LIN {X 0,Y 256.905,Z 476.365,A -85,B 0,C 180,E1 -19492.497,E2 -19492.497} C_VEL
LIN {X 0,Y 253.744,Z 490.842,A -85,B 0,C 180,E1 -19494.195,E2 -19494.195} C_VEL
LIN {X 0,Y 250.282,Z 505.582,A -85,B 0,C 180,E1 -19496.323,E2 -19496.323} C_VEL
LIN {X 0,Y 246.869,Z 518.814,A -85,B 0,C 180,E1 -19498.654,E2 -19498.654} C_VEL
LIN {X 0,Y 243.85,Z 530.517,A -85,B 0,C 180,E1 -19501.14,E2 -19501.14} C_VEL
LIN {X 0,Y 240.923,Z 541.947,A -85,B 0,C 180,E1 -19504.056,E2 -19504.056} C_VEL
LIN {X 0,Y 238.58,Z 551.642,A -85,B 0,C 180,E1 -19507.031,E2 -19507.031} C_VEL
LIN {X 0,Y 236.824,Z 559.89,A -85,B 0,C 180,E1 -19510.05,E2 -19510.05} C_VEL
LIN {X 0,Y 235.764,Z 565.839,A -85,B 0,C 180,E1 -19512.662,E2 -19512.662} C_VEL
LIN {X 0,Y 234.817,Z 572.47,A -85,B 0,C 180,E1 -19516.151,E2 -19516.151} C_VEL
LIN {X 0,Y 234.44,Z 577.709,A -85,B 0,C 180,E1 -19519.642,E2 -19519.642} C_VEL
LIN {X 0,Y 234.502,Z 581.558,A -85,B 0,C 180,E1 -19523.119,E2 -19523.119} C_VEL
LIN {X 0,Y 234.607,Z 584.124,A -85,B 0,C 180,E1 -19526.569,E2 -19526.569} C_VEL
LIN {X 0,Y 234.696,Z 584.956,A -85,B 0,C 180,E1 -19528.288,E2 -19528.288} C_VEL
LIN {X 0,Y 234.734,Z 585.482,A -85,B 0,C 180,E1 -19530.004,E2 -19530.004} C_VEL
LIN {X 0,Y 234.443,Z 585.509,A -85,B 0,C 180,E1 -19533.441,E2 -19533.441} C_VEL
LIN {X 0,Y 234.354,Z 585.124,A -85,B 0,C 180,E1 -19535.166,E2 -19535.166} C_VEL
LIN {X 0,Y 233.92,Z 583.497,A -85,B 0,C 180,E1 -19538.644,E2 -19538.644} C_VEL
LIN {X 0,Y 233.963,Z 580.814,A -85,B 0,C 180,E1 -19542.142,E2 -19542.142} C_VEL
LIN {X 0,Y 234.616,Z 577.208,A -85,B 0,C 180,E1 -19545.644,E2 -19545.644} C_VEL
LIN {X 0,Y 236.323,Z 571.284,A -85,B 0,C 180,E1 -19550.003,E2 -19550.003} C_VEL
LIN {X 0,Y 239.288,Z 563.871,A -85,B 0,C 180,E1 -19554.283,E2 -19554.283} C_VEL
LIN {X 0,Y 243.617,Z 554.947,A -85,B 0,C 180,E1 -19558.428,E2 -19558.428} C_VEL
LIN {X 0,Y 249.42,Z 544.436,A -85,B 0,C 180,E1 -19562.373,E2 -19562.373} C_VEL
LIN {X 0,Y 255.768,Z 533.545,A -85,B 0,C 180,E1 -19565.73,E2 -19565.73} C_VEL
LIN {X 0,Y 263.313,Z 521.165,A -85,B 0,C 180,E1 -19568.85,E2 -19568.85} C_VEL
LIN {X 0,Y 271.994,Z 507.097,A -85,B 0,C 180,E1 -19571.713,E2 -19571.713} C_VEL
LIN {X 0,Y 281.689,Z 491.098,A -85,B 0,C 180,E1 -19574.317,E2 -19574.317} C_VEL
LIN {X 0,Y 290.818,Z 473.344,A -85,B 0,C 180,E1 -19577.307,E2 -19577.307} C_VEL
LIN {X 0,Y 292.844,Z 469.182,A -85,B 0,C 180,E1 -19578.075,E2 -19578.075} C_VEL
LIN {X 0,Y 292.392,Z 467.764,A -85,B 0,C 180,E1 -19579.536,E2 -19579.536} C_VEL
LIN {X 0,Y 291.53,Z 467.553,A -85,B 0,C 180,E1 -19581.187,E2 -19581.187} C_VEL
LIN {X 0,Y 290.328,Z 468.711,A -85,B 0,C 180,E1 -19583.023,E2 -19583.023} C_VEL
LIN {X 0,Y 288.699,Z 471.49,A -85,B 0,C 180,E1 -19585.105,E2 -19585.105} C_VEL
LIN {X 0,Y 288.039,Z 472.753,A -85,B 0,C 180,E1 -19585.863,E2 -19585.863} C_VEL
LIN {X 0,Y 287.443,Z 473.689,A -85,B 0,C 180,E1 -19586.205,E2 -19586.205} C_VEL
LIN {X 0,Y 280.242,Z 483.352,A -85,B 0,C 180,E1 -19588.222,E2 -19588.222} C_VEL
LIN {X 0,Y 272.71,Z 492.785,A -85,B 0,C 180,E1 -19590.683,E2 -19590.683} C_VEL
LIN {X 0,Y 267.529,Z 498.863,A -85,B 0,C 180,E1 -19592.631,E2 -19592.631} C_VEL
LIN {X 0,Y 261.304,Z 505.728,A -85,B 0,C 180,E1 -19595.363,E2 -19595.363} C_VEL
LIN {X 0,Y 255.757,Z 511.304,A -85,B 0,C 180,E1 -19598.225,E2 -19598.225} C_VEL
LIN {X 0,Y 252.054,Z 514.612,A -85,B 0,C 180,E1 -19600.453,E2 -19600.453} C_VEL
LIN {X 0,Y 247.721,Z 517.909,A -85,B 0,C 180,E1 -19603.519,E2 -19603.519} C_VEL
LIN {X 0,Y 244.113,Z 519.898,A -85,B 0,C 180,E1 -19606.685,E2 -19606.685} C_VEL
LIN {X 0,Y 241.301,Z 520.551,A -85,B 0,C 180,E1 -19609.936,E2 -19609.936} C_VEL
LIN {X 0,Y 239.14,Z 519.825,A -85,B 0,C 180,E1 -19613.25,E2 -19613.25} C_VEL
LIN {X 0,Y 238.303,Z 518.908,A -85,B 0,C 180,E1 -19614.925,E2 -19614.925} C_VEL
LIN {X 0,Y 237.418,Z 517.65,A -85,B 0,C 180,E1 -19616.607,E2 -19616.607} C_VEL
LIN {X 0,Y 236.444,Z 513.942,A -85,B 0,C 180,E1 -19620.001,E2 -19620.001} C_VEL
LIN {X 0,Y 236.062,Z 508.652,A -85,B 0,C 180,E1 -19623.414,E2 -19623.414} C_VEL
LIN {X 0,Y 236.015,Z 503.521,A -85,B 0,C 180,E1 -19625.983,E2 -19625.983} C_VEL
LIN {X 0,Y 236.487,Z 495.93,A -85,B 0,C 180,E1 -19629.087,E2 -19629.087} C_VEL
LIN {X 0,Y 237.296,Z 487.239,A -85,B 0,C 180,E1 -19631.966,E2 -19631.966} C_VEL
LIN {X 0,Y 238.497,Z 476.352,A -85,B 0,C 180,E1 -19634.943,E2 -19634.943} C_VEL
LIN {X 0,Y 239.829,Z 465.148,A -85,B 0,C 180,E1 -19637.48,E2 -19637.48} C_VEL
LIN {X 0,Y 241.31,Z 454.184,A -85,B 0,C 180,E1 -19639.569,E2 -19639.569} C_VEL
LIN {X 0,Y 243.089,Z 439.84,A -85,B 0,C 180,E1 -19641.854,E2 -19641.854} C_VEL
LIN {X 0,Y 244.85,Z 423.851,A -85,B 0,C 180,E1 -19643.919,E2 -19643.919} C_VEL
LIN {X 0,Y 245.311,Z 420.209,A -85,B 0,C 180,E1 -19644.321,E2 -19644.321} C_VEL
LIN {X 0,Y 243.169,Z 407.684,A -85,B 0,C 180,E1 -19645.846,E2 -19645.846} C_VEL
LIN {X 0,Y 240.045,Z 393.035,A -85,B 0,C 180,E1 -19647.435,E2 -19647.435} C_VEL
LIN {X 0,Y 236.454,Z 377.897,A -85,B 0,C 180,E1 -19648.872,E2 -19648.872} C_VEL
LIN {X 0,Y 237.051,Z 372.231,A -85,B 0,C 180,E1 -19653.102,E2 -19653.102} C_VEL
LIN {X 0,Y 237.434,Z 368.102,A -85,B 0,C 180,E1 -19656.3,E2 -19656.3} C_VEL
LIN {X 0,Y 237.427,Z 366.543,A -85,B 0,C 180,E1 -19657.625,E2 -19657.625} C_VEL
LIN {X 0,Y 239.402,Z 369.891,A -85,B 0,C 180,E1 -19660.242,E2 -19660.242} C_VEL
LIN {X 0,Y 241.091,Z 374.148,A -85,B 0,C 180,E1 -19663.212,E2 -19663.212} C_VEL
LIN {X 0,Y 242.39,Z 380.678,A -85,B 0,C 180,E1 -19667.152,E2 -19667.152} C_VEL
LIN {X 0,Y 243.304,Z 386.405,A -85,B 0,C 180,E1 -19670.54,E2 -19670.54} C_VEL
LIN {X 0,Y 243.456,Z 389.408,A -85,B 0,C 180,E1 -19672.147,E2 -19672.147} C_VEL
LIN {X 0,Y 243.101,Z 397.462,A -85,B 0,C 180,E1 -19676.181,E2 -19676.181} C_VEL
LIN {X 0,Y 242.899,Z 404.228,A -85,B 0,C 180,E1 -19679.392,E2 -19679.392} C_VEL
LIN {X 0,Y 247.97,Z 416.97,A -85,B 0,C 180,E1 -19680.702,E2 -19680.702} C_VEL
LIN {X 0,Y 251.388,Z 428.049,A -85,B 0,C 180,E1 -19682,E2 -19682} C_VEL
LIN {X 0,Y 252.545,Z 432.8,A -85,B 0,C 180,E1 -19682.604,E2 -19682.604} C_VEL
LIN {X 0,Y 251.252,Z 444.342,A -85,B 0,C 180,E1 -19683.779,E2 -19683.779} C_VEL
LIN {X 0,Y 249.556,Z 455.455,A -85,B 0,C 180,E1 -19685.23,E2 -19685.23} C_VEL
LIN {X 0,Y 247.569,Z 466.219,A -85,B 0,C 180,E1 -19687.021,E2 -19687.021} C_VEL
LIN {X 0,Y 246.071,Z 474.012,A -85,B 0,C 180,E1 -19688.641,E2 -19688.641} C_VEL
LIN {X 0,Y 244.072,Z 482.139,A -85,B 0,C 180,E1 -19690.658,E2 -19690.658} C_VEL
LIN {X 0,Y 242.05,Z 490.033,A -85,B 0,C 180,E1 -19693.117,E2 -19693.117} C_VEL
LIN {X 0,Y 240.449,Z 496.348,A -85,B 0,C 180,E1 -19695.611,E2 -19695.611} C_VEL
LIN {X 0,Y 238.794,Z 501.412,A -85,B 0,C 180,E1 -19698.107,E2 -19698.107} C_VEL
LIN {X 0,Y 237.558,Z 505.313,A -85,B 0,C 180,E1 -19700.632,E2 -19700.632} C_VEL
LIN {X 0,Y 236.889,Z 508.146,A -85,B 0,C 180,E1 -19703.181,E2 -19703.181} C_VEL
LIN {X 0,Y 236.463,Z 509.533,A -85,B 0,C 180,E1 -19704.88,E2 -19704.88} C_VEL
LIN {X 0,Y 236.064,Z 511.09,A -85,B 0,C 180,E1 -19708.29,E2 -19708.29} C_VEL
LIN {X 0,Y 236,Z 511.318,A -85,B 0,C 180,E1 -19709.996,E2 -19709.996} C_VEL
LIN {X 0,Y 236.17,Z 510.561,A -85,B 0,C 180,E1 -19713.408,E2 -19713.408} C_VEL
LIN {X 0,Y 236.885,Z 508.275,A -85,B 0,C 180,E1 -19716.811,E2 -19716.811} C_VEL
LIN {X 0,Y 237.535,Z 505.493,A -85,B 0,C 180,E1 -19719.361,E2 -19719.361} C_VEL
LIN {X 0,Y 238.772,Z 501.65,A -85,B 0,C 180,E1 -19721.886,E2 -19721.886} C_VEL
LIN {X 0,Y 240.398,Z 496.65,A -85,B 0,C 180,E1 -19724.384,E2 -19724.384} C_VEL
LIN {X 0,Y 241.989,Z 490.397,A -85,B 0,C 180,E1 -19726.879,E2 -19726.879} C_VEL
LIN {X 0,Y 244.003,Z 482.585,A -85,B 0,C 180,E1 -19729.339,E2 -19729.339} C_VEL
LIN {X 0,Y 245.927,Z 474.575,A -85,B 0,C 180,E1 -19731.364,E2 -19731.364} C_VEL
LIN {X 0,Y 247.709,Z 465.828,A -85,B 0,C 180,E1 -19733.178,E2 -19733.178} C_VEL
LIN {X 0,Y 249.618,Z 454.949,A -85,B 0,C 180,E1 -19734.977,E2 -19734.977} C_VEL
LIN {X 0,Y 251.342,Z 444.115,A -85,B 0,C 180,E1 -19736.37,E2 -19736.37} C_VEL
LIN {X 0,Y 252.59,Z 433.78,A -85,B 0,C 180,E1 -19737.417,E2 -19737.417} C_VEL
LIN {X 0,Y 251.685,Z 429.238,A -85,B 0,C 180,E1 -19737.979,E2 -19737.979} C_VEL
LIN {X 0,Y 248.62,Z 418.97,A -85,B 0,C 180,E1 -19739.209,E2 -19739.209} C_VEL
LIN {X 0,Y 244.147,Z 407.043,A -85,B 0,C 180,E1 -19740.462,E2 -19740.462} C_VEL
LIN {X 0,Y 242.956,Z 404.156,A -85,B 0,C 180,E1 -19740.782,E2 -19740.782} C_VEL
LIN {X 0,Y 243.296,Z 394.738,A -85,B 0,C 180,E1 -19745.285,E2 -19745.285} C_VEL
LIN {X 0,Y 243.468,Z 388.645,A -85,B 0,C 180,E1 -19748.386,E2 -19748.386} C_VEL
LIN {X 0,Y 242.872,Z 383.713,A -85,B 0,C 180,E1 -19751.203,E2 -19751.203} C_VEL
LIN {X 0,Y 241.916,Z 378.028,A -85,B 0,C 180,E1 -19754.618,E2 -19754.618} C_VEL
LIN {X 0,Y 240.913,Z 372.705,A -85,B 0,C 180,E1 -19757.858,E2 -19757.858} C_VEL
LIN {X 0,Y 239.516,Z 366.53,A -85,B 0,C 180,E1 -19761.961,E2 -19761.961} C_VEL
LIN {X 0,Y 237.915,Z 360.81,A -85,B 0,C 180,E1 -19765.856,E2 -19765.856} C_VEL
LIN {X 0,Y 236.193,Z 355.497,A -85,B 0,C 180,E1 -19769.634,E2 -19769.634} C_VEL
LIN {X 0,Y 234.939,Z 351.525,A -85,B 0,C 180,E1 -19772.617,E2 -19772.617} C_VEL
LIN {X 0,Y 234.985,Z 351.514,A -85,B 0,C 180,E1 -19777.119,E2 -19777.119} C_VEL
LIN {X 0,Y 235.016,Z 351.51,A -85,B 0,C 180,E1 -19780.794,E2 -19780.794} C_VEL
LIN {X 0,Y 235.092,Z 351.505,A -85,B 0,C 180,E1 -19784.391,E2 -19784.391} C_VEL
LIN {X 0,Y 235.217,Z 351.484,A -85,B 0,C 180,E1 -19789.672,E2 -19789.672} C_VEL
LIN {X 0,Y 235.382,Z 351.479,A -85,B 0,C 180,E1 -19793.14,E2 -19793.14} C_VEL
LIN {X 0,Y 235.573,Z 351.455,A -85,B 0,C 180,E1 -19798.29,E2 -19798.29} C_VEL
LIN {X 0,Y 235.586,Z 351.437,A -85,B 0,C 180,E1 -19801.709,E2 -19801.709} C_VEL
LIN {X 0,Y 235.384,Z 351.475,A -85,B 0,C 180,E1 -19806.859,E2 -19806.859} C_VEL
LIN {X 0,Y 235.217,Z 351.5,A -85,B 0,C 180,E1 -19810.327,E2 -19810.327} C_VEL
LIN {X 0,Y 235.133,Z 351.62,A -85,B 0,C 180,E1 -19813.503,E2 -19813.503} C_VEL
LIN {X 0,Y 236.344,Z 356.522,A -85,B 0,C 180,E1 -19817.299,E2 -19817.299} C_VEL
LIN {X 0,Y 237.921,Z 362.673,A -85,B 0,C 180,E1 -19821.668,E2 -19821.668} C_VEL
LIN {X 0,Y 239.693,Z 369.451,A -85,B 0,C 180,E1 -19826.091,E2 -19826.091} C_VEL
LIN {X 0,Y 241.634,Z 377.004,A -85,B 0,C 180,E1 -19830.596,E2 -19830.596} C_VEL
LIN {X 0,Y 243.935,Z 385.536,A -85,B 0,C 180,E1 -19835.274,E2 -19835.274} C_VEL
LIN {X 0,Y 243.915,Z 388.145,A -85,B 0,C 180,E1 -19836.519,E2 -19836.519} C_VEL
LIN {X 0,Y 242.269,Z 392.897,A -85,B 0,C 180,E1 -19838.533,E2 -19838.533} C_VEL
LIN {X 0,Y 240.84,Z 396.809,A -85,B 0,C 180,E1 -19840.155,E2 -19840.155} C_VEL
LIN {X 0,Y 240.506,Z 399.631,A -85,B 0,C 180,E1 -19841.401,E2 -19841.401} C_VEL
LIN {X 0,Y 240.639,Z 400.533,A -85,B 0,C 180,E1 -19841.82,E2 -19841.82} C_VEL
LIN {X 0,Y 243.092,Z 409.192,A -85,B 0,C 180,E1 -19845.743,E2 -19845.743} C_VEL
LIN {X 0,Y 246.068,Z 416.929,A -85,B 0,C 180,E1 -19846.482,E2 -19846.482} C_VEL
LIN {X 0,Y 247.388,Z 433.311,A -85,B 0,C 180,E1 -19847.614,E2 -19847.614} C_VEL
LIN {X 0,Y 248.674,Z 450.528,A -85,B 0,C 180,E1 -19849.115,E2 -19849.115} C_VEL
LIN {X 0,Y 249.886,Z 467.196,A -85,B 0,C 180,E1 -19850.901,E2 -19850.901} C_VEL
LIN {X 0,Y 250.161,Z 476.141,A -85,B 0,C 180,E1 -19851.976,E2 -19851.976} C_VEL
LIN {X 0,Y 246.847,Z 491.074,A -85,B 0,C 180,E1 -19853.794,E2 -19853.794} C_VEL
LIN {X 0,Y 243.34,Z 505.617,A -85,B 0,C 180,E1 -19855.979,E2 -19855.979} C_VEL
LIN {X 0,Y 239.82,Z 518.892,A -85,B 0,C 180,E1 -19858.416,E2 -19858.416} C_VEL
LIN {X 0,Y 236.585,Z 531.126,A -85,B 0,C 180,E1 -19861.142,E2 -19861.142} C_VEL
LIN {X 0,Y 233.681,Z 542.281,A -85,B 0,C 180,E1 -19864.146,E2 -19864.146} C_VEL
LIN {X 0,Y 231.35,Z 551.748,A -85,B 0,C 180,E1 -19867.217,E2 -19867.217} C_VEL
LIN {X 0,Y 229.426,Z 560.909,A -85,B 0,C 180,E1 -19870.825,E2 -19870.825} C_VEL
LIN {X 0,Y 228.287,Z 567.377,A -85,B 0,C 180,E1 -19873.919,E2 -19873.919} C_VEL
LIN {X 0,Y 227.718,Z 572.033,A -85,B 0,C 180,E1 -19876.621,E2 -19876.621} C_VEL
LIN {X 0,Y 227.459,Z 577.083,A -85,B 0,C 180,E1 -19880.22,E2 -19880.22} C_VEL
LIN {X 0,Y 227.517,Z 579.962,A -85,B 0,C 180,E1 -19882.907,E2 -19882.907} C_VEL
LIN {X 0,Y 227.648,Z 582.685,A -85,B 0,C 180,E1 -19886.464,E2 -19886.464} C_VEL
LIN {X 0,Y 227.741,Z 583.579,A -85,B 0,C 180,E1 -19888.236,E2 -19888.236} C_VEL
LIN {X 0,Y 227.77,Z 584.109,A -85,B 0,C 180,E1 -19890.004,E2 -19890.004} C_VEL
LIN {X 0,Y 227.435,Z 584.256,A -85,B 0,C 180,E1 -19893.547,E2 -19893.547} C_VEL
LIN {X 0,Y 227.317,Z 583.935,A -85,B 0,C 180,E1 -19895.326,E2 -19895.326} C_VEL
LIN {X 0,Y 226.866,Z 582.358,A -85,B 0,C 180,E1 -19898.915,E2 -19898.915} C_VEL
LIN {X 0,Y 226.939,Z 579.83,A -85,B 0,C 180,E1 -19902.524,E2 -19902.524} C_VEL
LIN {X 0,Y 227.965,Z 575.214,A -85,B 0,C 180,E1 -19907.119,E2 -19907.119} C_VEL
LIN {X 0,Y 230.037,Z 569.3,A -85,B 0,C 180,E1 -19911.511,E2 -19911.511} C_VEL
LIN {X 0,Y 233.506,Z 561.84,A -85,B 0,C 180,E1 -19915.879,E2 -19915.879} C_VEL
LIN {X 0,Y 238.439,Z 552.932,A -85,B 0,C 180,E1 -19920.075,E2 -19920.075} C_VEL
LIN {X 0,Y 244.119,Z 543.618,A -85,B 0,C 180,E1 -19923.659,E2 -19923.659} C_VEL
LIN {X 0,Y 250.873,Z 533.031,A -85,B 0,C 180,E1 -19927.039,E2 -19927.039} C_VEL
LIN {X 0,Y 258.872,Z 521.045,A -85,B 0,C 180,E1 -19930.153,E2 -19930.153} C_VEL
LIN {X 0,Y 267.978,Z 507.491,A -85,B 0,C 180,E1 -19932.994,E2 -19932.994} C_VEL
LIN {X 0,Y 278.001,Z 492.2,A -85,B 0,C 180,E1 -19935.579,E2 -19935.579} C_VEL
LIN {X 0,Y 287.573,Z 475.666,A -85,B 0,C 180,E1 -19938.485,E2 -19938.485} C_VEL
LIN {X 0,Y 288.337,Z 474.174,A -85,B 0,C 180,E1 -19938.845,E2 -19938.845} C_VEL
LIN {X 0,Y 287.63,Z 473.234,A -85,B 0,C 180,E1 -19940.559,E2 -19940.559} C_VEL
LIN {X 0,Y 286.482,Z 473.83,A -85,B 0,C 180,E1 -19942.172,E2 -19942.172} C_VEL
LIN {X 0,Y 285.119,Z 475.37,A -85,B 0,C 180,E1 -19943.731,E2 -19943.731} C_VEL
LIN {X 0,Y 283.632,Z 477.641,A -85,B 0,C 180,E1 -19945.257,E2 -19945.257} C_VEL
LIN {X 0,Y 275.067,Z 488.02,A -85,B 0,C 180,E1 -19947.551,E2 -19947.551} C_VEL
LIN {X 0,Y 266.339,Z 497.79,A -85,B 0,C 180,E1 -19950.346,E2 -19950.346} C_VEL
LIN {X 0,Y 260.231,Z 504.152,A -85,B 0,C 180,E1 -19952.671,E2 -19952.671} C_VEL
LIN {X 0,Y 253.884,Z 510.25,A -85,B 0,C 180,E1 -19955.467,E2 -19955.467} C_VEL
LIN {X 0,Y 248.301,Z 515.08,A -85,B 0,C 180,E1 -19958.411,E2 -19958.411} C_VEL
LIN {X 0,Y 243.417,Z 518.68,A -85,B 0,C 180,E1 -19961.483,E2 -19961.483} C_VEL
LIN {X 0,Y 239.214,Z 521.024,A -85,B 0,C 180,E1 -19964.668,E2 -19964.668} C_VEL
LIN {X 0,Y 235.831,Z 522.038,A -85,B 0,C 180,E1 -19967.96,E2 -19967.96} C_VEL
LIN {X 0,Y 233.284,Z 521.715,A -85,B 0,C 180,E1 -19971.337,E2 -19971.337} C_VEL
LIN {X 0,Y 231.34,Z 520.014,A -85,B 0,C 180,E1 -19974.772,E2 -19974.772} C_VEL
LIN {X 0,Y 230.412,Z 518.642,A -85,B 0,C 180,E1 -19976.503,E2 -19976.503} C_VEL
LIN {X 0,Y 229.412,Z 514.712,A -85,B 0,C 180,E1 -19980.001,E2 -19980.001} C_VEL
LIN {X 0,Y 229.019,Z 510.704,A -85,B 0,C 180,E1 -19982.639,E2 -19982.639} C_VEL
LIN {X 0,Y 228.983,Z 505.751,A -85,B 0,C 180,E1 -19985.284,E2 -19985.284} C_VEL
LIN {X 0,Y 229.185,Z 498.642,A -85,B 0,C 180,E1 -19988.376,E2 -19988.376} C_VEL
LIN {X 0,Y 230.084,Z 490.109,A -85,B 0,C 180,E1 -19991.408,E2 -19991.408} C_VEL
LIN {X 0,Y 230.965,Z 481.065,A -85,B 0,C 180,E1 -19994.09,E2 -19994.09} C_VEL
LIN {X 0,Y 232.253,Z 470.488,A -85,B 0,C 180,E1 -19996.707,E2 -19996.707} C_VEL
LIN {X 0,Y 233.796,Z 457.973,A -85,B 0,C 180,E1 -19999.31,E2 -19999.31} C_VEL
LIN {X 0,Y 235.535,Z 445.648,A -85,B 0,C 180,E1 -20001.44,E2 -20001.44} C_VEL
LIN {X 0,Y 237.279,Z 431.014,A -85,B 0,C 180,E1 -20003.551,E2 -20003.551} C_VEL
LIN {X 0,Y 238.461,Z 420.905,A -85,B 0,C 180,E1 -20004.767,E2 -20004.767} C_VEL
LIN {X 0,Y 235.854,Z 406.113,A -85,B 0,C 180,E1 -20006.62,E2 -20006.62} C_VEL
LIN {X 0,Y 232.298,Z 390.022,A -85,B 0,C 180,E1 -20008.369,E2 -20008.369} C_VEL
LIN {X 0,Y 229.533,Z 378.312,A -85,B 0,C 180,E1 -20009.524,E2 -20009.524} C_VEL
LIN {X 0,Y 230.106,Z 373.294,A -85,B 0,C 180,E1 -20013.352,E2 -20013.352} C_VEL
LIN {X 0,Y 230.482,Z 369.036,A -85,B 0,C 180,E1 -20016.724,E2 -20016.724} C_VEL
LIN {X 0,Y 232.638,Z 372.21,A -85,B 0,C 180,E1 -20019.377,E2 -20019.377} C_VEL
LIN {X 0,Y 234.452,Z 376.349,A -85,B 0,C 180,E1 -20022.414,E2 -20022.414} C_VEL
LIN {X 0,Y 235.29,Z 379.832,A -85,B 0,C 180,E1 -20024.666,E2 -20024.666} C_VEL
LIN {X 0,Y 236.289,Z 385.317,A -85,B 0,C 180,E1 -20028.038,E2 -20028.038} C_VEL
LIN {X 0,Y 236.988,Z 391.196,A -85,B 0,C 180,E1 -20031.477,E2 -20031.477} C_VEL
LIN {X 0,Y 236.588,Z 399.414,A -85,B 0,C 180,E1 -20035.635,E2 -20035.635} C_VEL
LIN {X 0,Y 236.442,Z 405.515,A -85,B 0,C 180,E1 -20038.47,E2 -20038.47} C_VEL
LIN {X 0,Y 241.699,Z 418.579,A -85,B 0,C 180,E1 -20039.898,E2 -20039.898} C_VEL
LIN {X 0,Y 244.788,Z 428.658,A -85,B 0,C 180,E1 -20041.128,E2 -20041.128} C_VEL
LIN {X 0,Y 246.2,Z 434.288,A -85,B 0,C 180,E1 -20041.881,E2 -20041.881} C_VEL
LIN {X 0,Y 244.991,Z 445.264,A -85,B 0,C 180,E1 -20043.037,E2 -20043.037} C_VEL
LIN {X 0,Y 243.2,Z 456.522,A -85,B 0,C 180,E1 -20044.538,E2 -20044.538} C_VEL
LIN {X 0,Y 241.122,Z 467.29,A -85,B 0,C 180,E1 -20046.37,E2 -20046.37} C_VEL
LIN {X 0,Y 239.569,Z 475.081,A -85,B 0,C 180,E1 -20048.032,E2 -20048.032} C_VEL
LIN {X 0,Y 237.469,Z 483.212,A -85,B 0,C 180,E1 -20050.098,E2 -20050.098} C_VEL
LIN {X 0,Y 235.347,Z 491.108,A -85,B 0,C 180,E1 -20052.621,E2 -20052.621} C_VEL
LIN {X 0,Y 233.662,Z 497.424,A -85,B 0,C 180,E1 -20055.183,E2 -20055.183} C_VEL
LIN {X 0,Y 231.932,Z 502.489,A -85,B 0,C 180,E1 -20057.75,E2 -20057.75} C_VEL
LIN {X 0,Y 230.635,Z 506.391,A -85,B 0,C 180,E1 -20060.348,E2 -20060.348} C_VEL
LIN {X 0,Y 229.921,Z 509.224,A -85,B 0,C 180,E1 -20062.973,E2 -20062.973} C_VEL
LIN {X 0,Y 229.474,Z 510.61,A -85,B 0,C 180,E1 -20064.724,E2 -20064.724} C_VEL
LIN {X 0,Y 229.057,Z 512.166,A -85,B 0,C 180,E1 -20068.238,E2 -20068.238} C_VEL
LIN {X 0,Y 228.989,Z 512.394,A -85,B 0,C 180,E1 -20069.996,E2 -20069.996} C_VEL
LIN {X 0,Y 229.192,Z 511.634,A -85,B 0,C 180,E1 -20073.512,E2 -20073.512} C_VEL
LIN {X 0,Y 229.917,Z 509.351,A -85,B 0,C 180,E1 -20077.019,E2 -20077.019} C_VEL
LIN {X 0,Y 230.611,Z 506.568,A -85,B 0,C 180,E1 -20079.645,E2 -20079.645} C_VEL
LIN {X 0,Y 231.91,Z 502.724,A -85,B 0,C 180,E1 -20082.243,E2 -20082.243} C_VEL
LIN {X 0,Y 233.612,Z 497.723,A -85,B 0,C 180,E1 -20084.811,E2 -20084.811} C_VEL
LIN {X 0,Y 235.297,Z 491.466,A -85,B 0,C 180,E1 -20087.374,E2 -20087.374} C_VEL
LIN {X 0,Y 237.417,Z 483.65,A -85,B 0,C 180,E1 -20089.898,E2 -20089.898} C_VEL
LIN {X 0,Y 239.408,Z 475.641,A -85,B 0,C 180,E1 -20091.975,E2 -20091.975} C_VEL
LIN {X 0,Y 241.272,Z 466.891,A -85,B 0,C 180,E1 -20093.834,E2 -20093.834} C_VEL
LIN {X 0,Y 243.273,Z 456.005,A -85,B 0,C 180,E1 -20095.675,E2 -20095.675} C_VEL
LIN {X 0,Y 245.071,Z 445.155,A -85,B 0,C 180,E1 -20097.101,E2 -20097.101} C_VEL
LIN {X 0,Y 246.305,Z 434.831,A -85,B 0,C 180,E1 -20098.177,E2 -20098.177} C_VEL
LIN {X 0,Y 243.425,Z 423.902,A -85,B 0,C 180,E1 -20099.604,E2 -20099.604} C_VEL
LIN {X 0,Y 239.273,Z 412.202,A -85,B 0,C 180,E1 -20100.956,E2 -20100.956} C_VEL
LIN {X 0,Y 236.452,Z 405.271,A -85,B 0,C 180,E1 -20101.688,E2 -20101.688} C_VEL
LIN {X 0,Y 236.786,Z 396.656,A -85,B 0,C 180,E1 -20105.881,E2 -20105.881} C_VEL
LIN {X 0,Y 236.978,Z 391.551,A -85,B 0,C 180,E1 -20108.514,E2 -20108.514} C_VEL
LIN {X 0,Y 236.569,Z 387.535,A -85,B 0,C 180,E1 -20110.805,E2 -20110.805} C_VEL
LIN {X 0,Y 235.633,Z 381.717,A -85,B 0,C 180,E1 -20114.288,E2 -20114.288} C_VEL
LIN {X 0,Y 234.409,Z 375.054,A -85,B 0,C 180,E1 -20118.543,E2 -20118.543} C_VEL
LIN {X 0,Y 233.051,Z 368.735,A -85,B 0,C 180,E1 -20122.905,E2 -20122.905} C_VEL
LIN {X 0,Y 231.349,Z 363.014,A -85,B 0,C 180,E1 -20126.851,E2 -20126.851} C_VEL
LIN {X 0,Y 229.832,Z 357.949,A -85,B 0,C 180,E1 -20130.707,E2 -20130.707} C_VEL
LIN {X 0,Y 228.681,Z 354.842,A -85,B 0,C 180,E1 -20133.019,E2 -20133.019} C_VEL
LIN {X 0,Y 227.928,Z 352.405,A -85,B 0,C 180,E1 -20135.036,E2 -20135.036} C_VEL
LIN {X 0,Y 227.992,Z 352.39,A -85,B 0,C 180,E1 -20138.289,E2 -20138.289} C_VEL
LIN {X 0,Y 228.026,Z 352.389,A -85,B 0,C 180,E1 -20142.815,E2 -20142.815} C_VEL
LIN {X 0,Y 228.073,Z 352.384,A -85,B 0,C 180,E1 -20147.543,E2 -20147.543} C_VEL
LIN {X 0,Y 228.285,Z 352.345,A -85,B 0,C 180,E1 -20151.145,E2 -20151.145} C_VEL
LIN {X 0,Y 228.333,Z 352.356,A -85,B 0,C 180,E1 -20152.927,E2 -20152.927} C_VEL
LIN {X 0,Y 228.531,Z 352.332,A -85,B 0,C 180,E1 -20158.237,E2 -20158.237} C_VEL
LIN {X 0,Y 228.546,Z 352.314,A -85,B 0,C 180,E1 -20161.761,E2 -20161.761} C_VEL
LIN {X 0,Y 228.335,Z 352.353,A -85,B 0,C 180,E1 -20167.071,E2 -20167.071} C_VEL
LIN {X 0,Y 228.142,Z 352.379,A -85,B 0,C 180,E1 -20170.651,E2 -20170.651} C_VEL
LIN {X 0,Y 228.085,Z 352.428,A -85,B 0,C 180,E1 -20172.004,E2 -20172.004} C_VEL
LIN {X 0,Y 229.345,Z 357.387,A -85,B 0,C 180,E1 -20176.009,E2 -20176.009} C_VEL
LIN {X 0,Y 231.179,Z 364.737,A -85,B 0,C 180,E1 -20181.395,E2 -20181.395} C_VEL
LIN {X 0,Y 232.933,Z 371.561,A -85,B 0,C 180,E1 -20185.943,E2 -20185.943} C_VEL
LIN {X 0,Y 234.887,Z 379.168,A -85,B 0,C 180,E1 -20190.573,E2 -20190.573} C_VEL
LIN {X 0,Y 237.166,Z 387.619,A -85,B 0,C 180,E1 -20195.299,E2 -20195.299} C_VEL
LIN {X 0,Y 239.417,Z 396.14,A -85,B 0,C 180,E1 -20199.676,E2 -20199.676} C_VEL
LIN {X 0,Y 240.639,Z 400.533,A -85,B 0,C 180,E1 -20201.82,E2 -20201.82} C_VEL
LIN {X 0,Y 240.448,Z 402.594,A -85,B 0,C 180,E1 -20202.679,E2 -20202.679} C_VEL
LIN {X 0,Y 238.65,Z 406.687,A -85,B 0,C 180,E1 -20203.976,E2 -20203.976} C_VEL
LIN {X 0,Y 237.502,Z 410.566,A -85,B 0,C 180,E1 -20204.85,E2 -20204.85} C_VEL
LIN {X 0,Y 237.65,Z 413.876,A -85,B 0,C 180,E1 -20205.375,E2 -20205.375} C_VEL
LIN {X 0,Y 238.021,Z 415.018,A -85,B 0,C 180,E1 -20205.506,E2 -20205.506} C_VEL
LIN {X 0,Y 239.647,Z 419.2,A -85,B 0,C 180,E1 -20205.922,E2 -20205.922} C_VEL
LIN {X 0,Y 240.959,Z 436.294,A -85,B 0,C 180,E1 -20207.192,E2 -20207.192} C_VEL
LIN {X 0,Y 242.154,Z 453.884,A -85,B 0,C 180,E1 -20208.847,E2 -20208.847} C_VEL
LIN {X 0,Y 243.147,Z 469.57,A -85,B 0,C 180,E1 -20210.645,E2 -20210.645} C_VEL
LIN {X 0,Y 243.31,Z 476.685,A -85,B 0,C 180,E1 -20211.543,E2 -20211.543} C_VEL
LIN {X 0,Y 239.64,Z 492.5,A -85,B 0,C 180,E1 -20213.573,E2 -20213.573} C_VEL
LIN {X 0,Y 236.127,Z 506.658,A -85,B 0,C 180,E1 -20215.827,E2 -20215.827} C_VEL
LIN {X 0,Y 232.826,Z 518.686,A -85,B 0,C 180,E1 -20218.137,E2 -20218.137} C_VEL
LIN {X 0,Y 229.305,Z 531.596,A -85,B 0,C 180,E1 -20221.142,E2 -20221.142} C_VEL
LIN {X 0,Y 226.406,Z 542.522,A -85,B 0,C 180,E1 -20224.247,E2 -20224.247} C_VEL
LIN {X 0,Y 223.817,Z 552.993,A -85,B 0,C 180,E1 -20227.869,E2 -20227.869} C_VEL
LIN {X 0,Y 222.057,Z 561.967,A -85,B 0,C 180,E1 -20231.709,E2 -20231.709} C_VEL
LIN {X 0,Y 221.011,Z 568.616,A -85,B 0,C 180,E1 -20235.267,E2 -20235.267} C_VEL
LIN {X 0,Y 220.519,Z 574.137,A -85,B 0,C 180,E1 -20238.981,E2 -20238.981} C_VEL
LIN {X 0,Y 220.536,Z 578.336,A -85,B 0,C 180,E1 -20242.681,E2 -20242.681} C_VEL
LIN {X 0,Y 220.683,Z 581.184,A -85,B 0,C 180,E1 -20246.353,E2 -20246.353} C_VEL
LIN {X 0,Y 220.779,Z 582.102,A -85,B 0,C 180,E1 -20248.18,E2 -20248.18} C_VEL
LIN {X 0,Y 220.806,Z 582.707,A -85,B 0,C 180,E1 -20250.004,E2 -20250.004} C_VEL
LIN {X 0,Y 220.427,Z 582.989,A -85,B 0,C 180,E1 -20253.66,E2 -20253.66} C_VEL
LIN {X 0,Y 220.281,Z 582.696,A -85,B 0,C 180,E1 -20255.497,E2 -20255.497} C_VEL
LIN {X 0,Y 219.81,Z 581.218,A -85,B 0,C 180,E1 -20259.203,E2 -20259.203} C_VEL
LIN {X 0,Y 219.933,Z 578.814,A -85,B 0,C 180,E1 -20262.93,E2 -20262.93} C_VEL
LIN {X 0,Y 220.972,Z 574.614,A -85,B 0,C 180,E1 -20267.42,E2 -20267.42} C_VEL
LIN {X 0,Y 223.297,Z 568.645,A -85,B 0,C 180,E1 -20272.195,E2 -20272.195} C_VEL
LIN {X 0,Y 227.021,Z 561.468,A -85,B 0,C 180,E1 -20276.676,E2 -20276.676} C_VEL
LIN {X 0,Y 232.247,Z 552.904,A -85,B 0,C 180,E1 -20280.964,E2 -20280.964} C_VEL
LIN {X 0,Y 238.9,Z 542.918,A -85,B 0,C 180,E1 -20285.009,E2 -20285.009} C_VEL
LIN {X 0,Y 246.161,Z 532.68,A -85,B 0,C 180,E1 -20288.391,E2 -20288.391} C_VEL
LIN {X 0,Y 254.545,Z 521.139,A -85,B 0,C 180,E1 -20291.506,E2 -20291.506} C_VEL
LIN {X 0,Y 265.262,Z 506.533,A -85,B 0,C 180,E1 -20294.6,E2 -20294.6} C_VEL
LIN {X 0,Y 273.451,Z 495.147,A -85,B 0,C 180,E1 -20296.561,E2 -20296.561} C_VEL
LIN {X 0,Y 282.623,Z 480.996,A -85,B 0,C 180,E1 -20299.139,E2 -20299.139} C_VEL
LIN {X 0,Y 283.505,Z 479.12,A -85,B 0,C 180,E1 -20299.87,E2 -20299.87} C_VEL
LIN {X 0,Y 283.349,Z 478.942,A -85,B 0,C 180,E1 -20300.259,E2 -20300.259} C_VEL
LIN {X 0,Y 282.432,Z 479.11,A -85,B 0,C 180,E1 -20301.531,E2 -20301.531} C_VEL
LIN {X 0,Y 280.2,Z 481.172,A -85,B 0,C 180,E1 -20303.831,E2 -20303.831} C_VEL
LIN {X 0,Y 278.715,Z 482.901,A -85,B 0,C 180,E1 -20304.553,E2 -20304.553} C_VEL
LIN {X 0,Y 269.939,Z 492.533,A -85,B 0,C 180,E1 -20306.857,E2 -20306.857} C_VEL
LIN {X 0,Y 261.859,Z 500.725,A -85,B 0,C 180,E1 -20309.341,E2 -20309.341} C_VEL
LIN {X 0,Y 254.555,Z 507.568,A -85,B 0,C 180,E1 -20312.008,E2 -20312.008} C_VEL
LIN {X 0,Y 247.957,Z 513.201,A -85,B 0,C 180,E1 -20314.84,E2 -20314.84} C_VEL
LIN {X 0,Y 242.129,Z 517.617,A -85,B 0,C 180,E1 -20317.832,E2 -20317.832} C_VEL
LIN {X 0,Y 237.022,Z 520.851,A -85,B 0,C 180,E1 -20320.965,E2 -20320.965} C_VEL
LIN {X 0,Y 232.614,Z 522.894,A -85,B 0,C 180,E1 -20324.222,E2 -20324.222} C_VEL
LIN {X 0,Y 229.08,Z 523.638,A -85,B 0,C 180,E1 -20327.6,E2 -20327.6} C_VEL
LIN {X 0,Y 226.397,Z 523.045,A -85,B 0,C 180,E1 -20331.071,E2 -20331.071} C_VEL
LIN {X 0,Y 224.372,Z 521.093,A -85,B 0,C 180,E1 -20334.609,E2 -20334.609} C_VEL
LIN {X 0,Y 223.406,Z 519.606,A -85,B 0,C 180,E1 -20336.393,E2 -20336.393} C_VEL
LIN {X 0,Y 222.36,Z 515.422,A -85,B 0,C 180,E1 -20340.001,E2 -20340.001} C_VEL
LIN {X 0,Y 221.945,Z 509.619,A -85,B 0,C 180,E1 -20343.632,E2 -20343.632} C_VEL
LIN {X 0,Y 221.891,Z 503.141,A -85,B 0,C 180,E1 -20346.822,E2 -20346.822} C_VEL
LIN {X 0,Y 222.524,Z 495.171,A -85,B 0,C 180,E1 -20350.004,E2 -20350.004} C_VEL
LIN {X 0,Y 223.366,Z 486.965,A -85,B 0,C 180,E1 -20352.724,E2 -20352.724} C_VEL
LIN {X 0,Y 224.493,Z 477.318,A -85,B 0,C 180,E1 -20355.433,E2 -20355.433} C_VEL
LIN {X 0,Y 225.932,Z 465.899,A -85,B 0,C 180,E1 -20358.124,E2 -20358.124} C_VEL
LIN {X 0,Y 227.521,Z 454.723,A -85,B 0,C 180,E1 -20360.336,E2 -20360.336} C_VEL
LIN {X 0,Y 229.233,Z 441.633,A -85,B 0,C 180,E1 -20362.535,E2 -20362.535} C_VEL
LIN {X 0,Y 231.047,Z 426.13,A -85,B 0,C 180,E1 -20364.677,E2 -20364.677} C_VEL
LIN {X 0,Y 231.582,Z 422.215,A -85,B 0,C 180,E1 -20365.143,E2 -20365.143} C_VEL
LIN {X 0,Y 229.404,Z 409.226,A -85,B 0,C 180,E1 -20366.833,E2 -20366.833} C_VEL
LIN {X 0,Y 226.036,Z 393.427,A -85,B 0,C 180,E1 -20368.661,E2 -20368.661} C_VEL
LIN {X 0,Y 222.643,Z 378.76,A -85,B 0,C 180,E1 -20370.159,E2 -20370.159} C_VEL
LIN {X 0,Y 223.311,Z 373.187,A -85,B 0,C 180,E1 -20374.507,E2 -20374.507} C_VEL
LIN {X 0,Y 223.531,Z 371.665,A -85,B 0,C 180,E1 -20375.896,E2 -20375.896} C_VEL
LIN {X 0,Y 226.117,Z 375.146,A -85,B 0,C 180,E1 -20379.005,E2 -20379.005} C_VEL
LIN {X 0,Y 227.861,Z 378.786,A -85,B 0,C 180,E1 -20381.711,E2 -20381.711} C_VEL
LIN {X 0,Y 228.697,Z 381.683,A -85,B 0,C 180,E1 -20383.745,E2 -20383.745} C_VEL
LIN {X 0,Y 229.83,Z 387.991,A -85,B 0,C 180,E1 -20387.716,E2 -20387.716} C_VEL
LIN {X 0,Y 230.463,Z 393.126,A -85,B 0,C 180,E1 -20390.74,E2 -20390.74} C_VEL
LIN {X 0,Y 230.222,Z 399.365,A -85,B 0,C 180,E1 -20394.025,E2 -20394.025} C_VEL
LIN {X 0,Y 229.896,Z 406.339,A -85,B 0,C 180,E1 -20397.455,E2 -20397.455} C_VEL
LIN {X 0,Y 235.186,Z 419.544,A -85,B 0,C 180,E1 -20398.965,E2 -20398.965} C_VEL
LIN {X 0,Y 238.228,Z 429.259,A -85,B 0,C 180,E1 -20400.208,E2 -20400.208} C_VEL
LIN {X 0,Y 239.985,Z 436.812,A -85,B 0,C 180,E1 -20401.251,E2 -20401.251} C_VEL
LIN {X 0,Y 238.367,Z 448.995,A -85,B 0,C 180,E1 -20402.6,E2 -20402.6} C_VEL
LIN {X 0,Y 236.667,Z 458.945,A -85,B 0,C 180,E1 -20404.019,E2 -20404.019} C_VEL
LIN {X 0,Y 234.466,Z 469.39,A -85,B 0,C 180,E1 -20405.891,E2 -20405.891} C_VEL
LIN {X 0,Y 232.652,Z 477.875,A -85,B 0,C 180,E1 -20407.811,E2 -20407.811} C_VEL
LIN {X 0,Y 230.885,Z 484.286,A -85,B 0,C 180,E1 -20409.505,E2 -20409.505} C_VEL
LIN {X 0,Y 228.659,Z 492.184,A -85,B 0,C 180,E1 -20412.096,E2 -20412.096} C_VEL
LIN {X 0,Y 226.888,Z 498.5,A -85,B 0,C 180,E1 -20414.73,E2 -20414.73} C_VEL
LIN {X 0,Y 225.08,Z 503.566,A -85,B 0,C 180,E1 -20417.371,E2 -20417.371} C_VEL
LIN {X 0,Y 223.717,Z 507.469,A -85,B 0,C 180,E1 -20420.046,E2 -20420.046} C_VEL
LIN {X 0,Y 222.958,Z 510.301,A -85,B 0,C 180,E1 -20422.752,E2 -20422.752} C_VEL
LIN {X 0,Y 222.509,Z 511.684,A -85,B 0,C 180,E1 -20424.558,E2 -20424.558} C_VEL
LIN {X 0,Y 222.049,Z 513.242,A -85,B 0,C 180,E1 -20428.182,E2 -20428.182} C_VEL
LIN {X 0,Y 221.976,Z 513.471,A -85,B 0,C 180,E1 -20429.996,E2 -20429.996} C_VEL
LIN {X 0,Y 222.211,Z 512.707,A -85,B 0,C 180,E1 -20433.622,E2 -20433.622} C_VEL
LIN {X 0,Y 222.952,Z 510.427,A -85,B 0,C 180,E1 -20437.239,E2 -20437.239} C_VEL
LIN {X 0,Y 223.693,Z 507.644,A -85,B 0,C 180,E1 -20439.946,E2 -20439.946} C_VEL
LIN {X 0,Y 225.057,Z 503.798,A -85,B 0,C 180,E1 -20442.622,E2 -20442.622} C_VEL
LIN {X 0,Y 226.842,Z 498.794,A -85,B 0,C 180,E1 -20445.264,E2 -20445.264} C_VEL
LIN {X 0,Y 228.626,Z 492.535,A -85,B 0,C 180,E1 -20447.898,E2 -20447.898} C_VEL
LIN {X 0,Y 230.835,Z 484.719,A -85,B 0,C 180,E1 -20450.49,E2 -20450.49} C_VEL
LIN {X 0,Y 232.937,Z 476.704,A -85,B 0,C 180,E1 -20452.619,E2 -20452.619} C_VEL
LIN {X 0,Y 234.868,Z 467.953,A -85,B 0,C 180,E1 -20454.526,E2 -20454.526} C_VEL
LIN {X 0,Y 236.965,Z 457.061,A -85,B 0,C 180,E1 -20456.41,E2 -20456.41} C_VEL
LIN {X 0,Y 238.858,Z 446.195,A -85,B 0,C 180,E1 -20457.867,E2 -20457.867} C_VEL
LIN {X 0,Y 240.09,Z 437.039,A -85,B 0,C 180,E1 -20458.843,E2 -20458.843} C_VEL
LIN {X 0,Y 237.358,Z 426.221,A -85,B 0,C 180,E1 -20460.327,E2 -20460.327} C_VEL
LIN {X 0,Y 233.408,Z 414.771,A -85,B 0,C 180,E1 -20461.745,E2 -20461.745} C_VEL
LIN {X 0,Y 229.96,Z 406.25,A -85,B 0,C 180,E1 -20462.712,E2 -20462.712} C_VEL
LIN {X 0,Y 230.292,Z 398.615,A -85,B 0,C 180,E1 -20466.492,E2 -20466.492} C_VEL
LIN {X 0,Y 230.469,Z 393.427,A -85,B 0,C 180,E1 -20469.247,E2 -20469.247} C_VEL
LIN {X 0,Y 229.708,Z 387.524,A -85,B 0,C 180,E1 -20472.752,E2 -20472.752} C_VEL
LIN {X 0,Y 228.775,Z 381.916,A -85,B 0,C 180,E1 -20476.274,E2 -20476.274} C_VEL
LIN {X 0,Y 227.573,Z 375.578,A -85,B 0,C 180,E1 -20480.531,E2 -20480.531} C_VEL
LIN {X 0,Y 226.479,Z 370.912,A -85,B 0,C 180,E1 -20483.871,E2 -20483.871} C_VEL
LIN {X 0,Y 224.849,Z 365.378,A -85,B 0,C 180,E1 -20487.902,E2 -20487.902} C_VEL
LIN {X 0,Y 223.793,Z 361.588,A -85,B 0,C 180,E1 -20490.872,E2 -20490.872} C_VEL
LIN {X 0,Y 222.17,Z 356.895,A -85,B 0,C 180,E1 -20494.719,E2 -20494.719} C_VEL
LIN {X 0,Y 220.977,Z 353.525,A -85,B 0,C 180,E1 -20497.809,E2 -20497.809} C_VEL
LIN {X 0,Y 220.928,Z 353.272,A -85,B 0,C 180,E1 -20498.541,E2 -20498.541} C_VEL
LIN {X 0,Y 221.005,Z 353.27,A -85,B 0,C 180,E1 -20503.369,E2 -20503.369} C_VEL
LIN {X 0,Y 221.092,Z 353.249,A -85,B 0,C 180,E1 -20509.004,E2 -20509.004} C_VEL
LIN {X 0,Y 221.284,Z 353.233,A -85,B 0,C 180,E1 -20512.701,E2 -20512.701} C_VEL
LIN {X 0,Y 221.489,Z 353.209,A -85,B 0,C 180,E1 -20518.181,E2 -20518.181} C_VEL
LIN {X 0,Y 221.504,Z 353.191,A -85,B 0,C 180,E1 -20521.818,E2 -20521.818} C_VEL
LIN {X 0,Y 221.286,Z 353.232,A -85,B 0,C 180,E1 -20527.298,E2 -20527.298} C_VEL
LIN {X 0,Y 221.145,Z 353.448,A -85,B 0,C 180,E1 -20530.631,E2 -20530.631} C_VEL
LIN {X 0,Y 222.578,Z 359.377,A -85,B 0,C 180,E1 -20535.568,E2 -20535.568} C_VEL
LIN {X 0,Y 224.399,Z 366.759,A -85,B 0,C 180,E1 -20541.11,E2 -20541.11} C_VEL
LIN {X 0,Y 226.156,Z 373.63,A -85,B 0,C 180,E1 -20545.789,E2 -20545.789} C_VEL
LIN {X 0,Y 228.046,Z 380.971,A -85,B 0,C 180,E1 -20550.366,E2 -20550.366} C_VEL
LIN {X 0,Y 230.419,Z 389.796,A -85,B 0,C 180,E1 -20555.416,E2 -20555.416} C_VEL
LIN {X 0,Y 232.885,Z 399.128,A -85,B 0,C 180,E1 -20560.299,E2 -20560.299} C_VEL
LIN {X 0,Y 235.553,Z 408.59,A -85,B 0,C 180,E1 -20564.866,E2 -20564.866} C_VEL
LIN {X 0,Y 238.021,Z 415.018,A -85,B 0,C 180,E1 -20565.506,E2 -20565.506} C_VEL
LIN {X 0,Y 238.504,Z 418.068,A -85,B 0,C 180,E1 -20565.731,E2 -20565.731} C_VEL
LIN {X 0,Y 237.616,Z 422.57,A -85,B 0,C 180,E1 -20565.9,E2 -20565.9} C_VEL
LIN {X 0,Y 234.548,Z 431.67,A -85,B 0,C 180,E1 -20566.189,E2 -20566.189} C_VEL
LIN {X 0,Y 234.246,Z 435.609,A -85,B 0,C 180,E1 -20566.46,E2 -20566.46} C_VEL
LIN {X 0,Y 235.331,Z 452.748,A -85,B 0,C 180,E1 -20568.12,E2 -20568.12} C_VEL
LIN {X 0,Y 236.283,Z 468.806,A -85,B 0,C 180,E1 -20570.009,E2 -20570.009} C_VEL
LIN {X 0,Y 236.383,Z 477.367,A -85,B 0,C 180,E1 -20571.131,E2 -20571.131} C_VEL
LIN {X 0,Y 232.78,Z 492.326,A -85,B 0,C 180,E1 -20573.132,E2 -20573.132} C_VEL
LIN {X 0,Y 229.221,Z 506.344,A -85,B 0,C 180,E1 -20575.45,E2 -20575.45} C_VEL
LIN {X 0,Y 225.624,Z 519.201,A -85,B 0,C 180,E1 -20578.032,E2 -20578.032} C_VEL
LIN {X 0,Y 222.533,Z 530.206,A -85,B 0,C 180,E1 -20580.697,E2 -20580.697} C_VEL
LIN {X 0,Y 219.567,Z 541.091,A -85,B 0,C 180,E1 -20583.866,E2 -20583.866} C_VEL
LIN {X 0,Y 217.177,Z 550.446,A -85,B 0,C 180,E1 -20587.155,E2 -20587.155} C_VEL
LIN {X 0,Y 215.317,Z 559.341,A -85,B 0,C 180,E1 -20590.955,E2 -20590.955} C_VEL
LIN {X 0,Y 214.131,Z 566.557,A -85,B 0,C 180,E1 -20594.783,E2 -20594.783} C_VEL
LIN {X 0,Y 213.55,Z 572.293,A -85,B 0,C 180,E1 -20598.616,E2 -20598.616} C_VEL
LIN {X 0,Y 213.524,Z 575.186,A -85,B 0,C 180,E1 -20600.901,E2 -20600.901} C_VEL
LIN {X 0,Y 213.532,Z 576.791,A -85,B 0,C 180,E1 -20602.44,E2 -20602.44} C_VEL
LIN {X 0,Y 213.712,Z 579.624,A -85,B 0,C 180,E1 -20606.234,E2 -20606.234} C_VEL
LIN {X 0,Y 213.817,Z 580.6,A -85,B 0,C 180,E1 -20608.121,E2 -20608.121} C_VEL
LIN {X 0,Y 213.869,Z 581.291,A -85,B 0,C 180,E1 -20610.005,E2 -20610.005} C_VEL
LIN {X 0,Y 213.428,Z 581.658,A -85,B 0,C 180,E1 -20613.781,E2 -20613.781} C_VEL
LIN {X 0,Y 213.245,Z 581.394,A -85,B 0,C 180,E1 -20615.679,E2 -20615.679} C_VEL
LIN {X 0,Y 212.766,Z 580.077,A -85,B 0,C 180,E1 -20619.511,E2 -20619.511} C_VEL
LIN {X 0,Y 212.917,Z 577.747,A -85,B 0,C 180,E1 -20623.364,E2 -20623.364} C_VEL
LIN {X 0,Y 213.955,Z 574.04,A -85,B 0,C 180,E1 -20627.715,E2 -20627.715} C_VEL
LIN {X 0,Y 215.969,Z 569.259,A -85,B 0,C 180,E1 -20631.981,E2 -20631.981} C_VEL
LIN {X 0,Y 219.644,Z 562.611,A -85,B 0,C 180,E1 -20636.617,E2 -20636.617} C_VEL
LIN {X 0,Y 224.863,Z 554.656,A -85,B 0,C 180,E1 -20641.049,E2 -20641.049} C_VEL
LIN {X 0,Y 231.611,Z 545.366,A -85,B 0,C 180,E1 -20645.212,E2 -20645.212} C_VEL
LIN {X 0,Y 239.768,Z 534.703,A -85,B 0,C 180,E1 -20649.069,E2 -20649.069} C_VEL
LIN {X 0,Y 248.415,Z 523.861,A -85,B 0,C 180,E1 -20652.22,E2 -20652.22} C_VEL
LIN {X 0,Y 259.302,Z 510.244,A -85,B 0,C 180,E1 -20655.359,E2 -20655.359} C_VEL
LIN {X 0,Y 270.074,Z 496.485,A -85,B 0,C 180,E1 -20657.875,E2 -20657.875} C_VEL
LIN {X 0,Y 278.589,Z 484.738,A -85,B 0,C 180,E1 -20660.108,E2 -20660.108} C_VEL
LIN {X 0,Y 278.271,Z 484.458,A -85,B 0,C 180,E1 -20660.847,E2 -20660.847} C_VEL
LIN {X 0,Y 276.71,Z 485.313,A -85,B 0,C 180,E1 -20662.443,E2 -20662.443} C_VEL
LIN {X 0,Y 276.062,Z 485.87,A -85,B 0,C 180,E1 -20663.064,E2 -20663.064} C_VEL
LIN {X 0,Y 275.261,Z 486.663,A -85,B 0,C 180,E1 -20663.491,E2 -20663.491} C_VEL
LIN {X 0,Y 263.757,Z 498.039,A -85,B 0,C 180,E1 -20666.435,E2 -20666.435} C_VEL
LIN {X 0,Y 254.516,Z 506.308,A -85,B 0,C 180,E1 -20669.281,E2 -20669.281} C_VEL
LIN {X 0,Y 247.155,Z 512.327,A -85,B 0,C 180,E1 -20672.019,E2 -20672.019} C_VEL
LIN {X 0,Y 241.734,Z 516.366,A -85,B 0,C 180,E1 -20674.333,E2 -20674.333} C_VEL
LIN {X 0,Y 235.973,Z 520.17,A -85,B 0,C 180,E1 -20677.222,E2 -20677.222} C_VEL
LIN {X 0,Y 230.648,Z 523.056,A -85,B 0,C 180,E1 -20680.417,E2 -20680.417} C_VEL
LIN {X 0,Y 226.041,Z 524.769,A -85,B 0,C 180,E1 -20683.751,E2 -20683.751} C_VEL
LIN {X 0,Y 222.33,Z 525.215,A -85,B 0,C 180,E1 -20687.217,E2 -20687.217} C_VEL
LIN {X 0,Y 219.52,Z 524.359,A -85,B 0,C 180,E1 -20690.789,E2 -20690.789} C_VEL
LIN {X 0,Y 217.399,Z 522.129,A -85,B 0,C 180,E1 -20694.435,E2 -20694.435} C_VEL
LIN {X 0,Y 216.065,Z 519.527,A -85,B 0,C 180,E1 -20697.204,E2 -20697.204} C_VEL
LIN {X 0,Y 215.084,Z 514.724,A -85,B 0,C 180,E1 -20700.937,E2 -20700.937} C_VEL
LIN {X 0,Y 214.863,Z 508.251,A -85,B 0,C 180,E1 -20704.691,E2 -20704.691} C_VEL
LIN {X 0,Y 214.953,Z 501.125,A -85,B 0,C 180,E1 -20707.988,E2 -20707.988} C_VEL
LIN {X 0,Y 215.87,Z 492.479,A -85,B 0,C 180,E1 -20711.265,E2 -20711.265} C_VEL
LIN {X 0,Y 216.911,Z 481.929,A -85,B 0,C 180,E1 -20714.544,E2 -20714.544} C_VEL
LIN {X 0,Y 218.308,Z 471.176,A -85,B 0,C 180,E1 -20717.325,E2 -20717.325} C_VEL
LIN {X 0,Y 219.973,Z 458.471,A -85,B 0,C 180,E1 -20720.088,E2 -20720.088} C_VEL
LIN {X 0,Y 221.681,Z 447.283,A -85,B 0,C 180,E1 -20722.116,E2 -20722.116} C_VEL
LIN {X 0,Y 223.539,Z 432.474,A -85,B 0,C 180,E1 -20724.372,E2 -20724.372} C_VEL
LIN {X 0,Y 224.66,Z 422,A -85,B 0,C 180,E1 -20725.726,E2 -20725.726} C_VEL
LIN {X 0,Y 221.923,Z 406.647,A -85,B 0,C 180,E1 -20727.773,E2 -20727.773} C_VEL
LIN {X 0,Y 217.901,Z 388.403,A -85,B 0,C 180,E1 -20729.88,E2 -20729.88} C_VEL
LIN {X 0,Y 215.727,Z 379.182,A -85,B 0,C 180,E1 -20730.854,E2 -20730.854} C_VEL
LIN {X 0,Y 216.4,Z 374.459,A -85,B 0,C 180,E1 -20734.777,E2 -20734.777} C_VEL
LIN {X 0,Y 218.906,Z 377.19,A -85,B 0,C 180,E1 -20737.59,E2 -20737.59} C_VEL
LIN {X 0,Y 221.079,Z 380.884,A -85,B 0,C 180,E1 -20740.668,E2 -20740.668} C_VEL
LIN {X 0,Y 222.339,Z 384.58,A -85,B 0,C 180,E1 -20743.358,E2 -20743.358} C_VEL
LIN {X 0,Y 223.463,Z 391.075,A -85,B 0,C 180,E1 -20747.55,E2 -20747.55} C_VEL
LIN {X 0,Y 224.034,Z 396.09,A -85,B 0,C 180,E1 -20750.565,E2 -20750.565} C_VEL
LIN {X 0,Y 223.712,Z 403.182,A -85,B 0,C 180,E1 -20754.317,E2 -20754.317} C_VEL
LIN {X 0,Y 223.485,Z 407.422,A -85,B 0,C 180,E1 -20756.401,E2 -20756.401} C_VEL
LIN {X 0,Y 228.754,Z 420.584,A -85,B 0,C 180,E1 -20757.986,E2 -20757.986} C_VEL
LIN {X 0,Y 231.842,Z 430.264,A -85,B 0,C 180,E1 -20759.291,E2 -20759.291} C_VEL
LIN {X 0,Y 233.743,Z 437.886,A -85,B 0,C 180,E1 -20760.409,E2 -20760.409} C_VEL
LIN {X 0,Y 232.157,Z 450.041,A -85,B 0,C 180,E1 -20761.801,E2 -20761.801} C_VEL
LIN {X 0,Y 230.378,Z 460.012,A -85,B 0,C 180,E1 -20763.254,E2 -20763.254} C_VEL
LIN {X 0,Y 228.086,Z 470.459,A -85,B 0,C 180,E1 -20765.172,E2 -20765.172} C_VEL
LIN {X 0,Y 226.171,Z 478.947,A -85,B 0,C 180,E1 -20767.139,E2 -20767.139} C_VEL
LIN {X 0,Y 223.92,Z 486.788,A -85,B 0,C 180,E1 -20769.319,E2 -20769.319} C_VEL
LIN {X 0,Y 221.586,Z 494.685,A -85,B 0,C 180,E1 -20772.086,E2 -20772.086} C_VEL
LIN {X 0,Y 220.129,Z 499.576,A -85,B 0,C 180,E1 -20774.249,E2 -20774.249} C_VEL
LIN {X 0,Y 218.238,Z 504.643,A -85,B 0,C 180,E1 -20776.968,E2 -20776.968} C_VEL
LIN {X 0,Y 216.806,Z 508.546,A -85,B 0,C 180,E1 -20779.726,E2 -20779.726} C_VEL
LIN {X 0,Y 215.998,Z 511.378,A -85,B 0,C 180,E1 -20782.517,E2 -20782.517} C_VEL
LIN {X 0,Y 215.542,Z 512.758,A -85,B 0,C 180,E1 -20784.382,E2 -20784.382} C_VEL
LIN {X 0,Y 215.04,Z 514.319,A -85,B 0,C 180,E1 -20788.123,E2 -20788.123} C_VEL
LIN {X 0,Y 214.962,Z 514.547,A -85,B 0,C 180,E1 -20789.995,E2 -20789.995} C_VEL
LIN {X 0,Y 215.228,Z 513.78,A -85,B 0,C 180,E1 -20793.74,E2 -20793.74} C_VEL
LIN {X 0,Y 215.562,Z 512.834,A -85,B 0,C 180,E1 -20795.608,E2 -20795.608} C_VEL
LIN {X 0,Y 215.991,Z 511.503,A -85,B 0,C 180,E1 -20797.474,E2 -20797.474} C_VEL
LIN {X 0,Y 216.782,Z 508.72,A -85,B 0,C 180,E1 -20800.266,E2 -20800.266} C_VEL
LIN {X 0,Y 218.214,Z 504.872,A -85,B 0,C 180,E1 -20803.024,E2 -20803.024} C_VEL
LIN {X 0,Y 220.087,Z 499.866,A -85,B 0,C 180,E1 -20805.744,E2 -20805.744} C_VEL
LIN {X 0,Y 221.961,Z 493.605,A -85,B 0,C 180,E1 -20808.454,E2 -20808.454} C_VEL
LIN {X 0,Y 224.274,Z 485.788,A -85,B 0,C 180,E1 -20811.118,E2 -20811.118} C_VEL
LIN {X 0,Y 226.476,Z 477.771,A -85,B 0,C 180,E1 -20813.302,E2 -20813.302} C_VEL
LIN {X 0,Y 228.26,Z 470.054,A -85,B 0,C 180,E1 -20815.041,E2 -20815.041} C_VEL
LIN {X 0,Y 230.508,Z 459.475,A -85,B 0,C 180,E1 -20816.965,E2 -20816.965} C_VEL
LIN {X 0,Y 232.446,Z 448.733,A -85,B 0,C 180,E1 -20818.488,E2 -20818.488} C_VEL
LIN {X 0,Y 233.788,Z 438.109,A -85,B 0,C 180,E1 -20819.697,E2 -20819.697} C_VEL
LIN {X 0,Y 230.829,Z 426.831,A -85,B 0,C 180,E1 -20821.325,E2 -20821.325} C_VEL
LIN {X 0,Y 226.721,Z 415.106,A -85,B 0,C 180,E1 -20822.835,E2 -20822.835} C_VEL
LIN {X 0,Y 223.565,Z 407.365,A -85,B 0,C 180,E1 -20823.747,E2 -20823.747} C_VEL
LIN {X 0,Y 224.041,Z 398.376,A -85,B 0,C 180,E1 -20828.349,E2 -20828.349} C_VEL
LIN {X 0,Y 224.008,Z 395.353,A -85,B 0,C 180,E1 -20830.016,E2 -20830.016} C_VEL
LIN {X 0,Y 223.091,Z 389.042,A -85,B 0,C 180,E1 -20833.866,E2 -20833.866} C_VEL
LIN {X 0,Y 222.012,Z 382.327,A -85,B 0,C 180,E1 -20838.334,E2 -20838.334} C_VEL
LIN {X 0,Y 220.731,Z 376.078,A -85,B 0,C 180,E1 -20842.774,E2 -20842.774} C_VEL
LIN {X 0,Y 219.466,Z 371.249,A -85,B 0,C 180,E1 -20846.357,E2 -20846.357} C_VEL
LIN {X 0,Y 218.543,Z 367.774,A -85,B 0,C 180,E1 -20849.033,E2 -20849.033} C_VEL
LIN {X 0,Y 216.983,Z 362.881,A -85,B 0,C 180,E1 -20853.034,E2 -20853.034} C_VEL
LIN {X 0,Y 215.499,Z 358.856,A -85,B 0,C 180,E1 -20856.961,E2 -20856.961} C_VEL
LIN {X 0,Y 214.31,Z 355.919,A -85,B 0,C 180,E1 -20859.858,E2 -20859.858} C_VEL
LIN {X 0,Y 213.898,Z 354.138,A -85,B 0,C 180,E1 -20861.471,E2 -20861.471} C_VEL
LIN {X 0,Y 213.916,Z 354.138,A -85,B 0,C 180,E1 -20864.761,E2 -20864.761} C_VEL
LIN {X 0,Y 214.12,Z 354.109,A -85,B 0,C 180,E1 -20869.924,E2 -20869.924} C_VEL
LIN {X 0,Y 214.219,Z 354.11,A -85,B 0,C 180,E1 -20872.459,E2 -20872.459} C_VEL
LIN {X 0,Y 214.423,Z 354.089,A -85,B 0,C 180,E1 -20878.121,E2 -20878.121} C_VEL
LIN {X 0,Y 214.462,Z 354.068,A -85,B 0,C 180,E1 -20881.877,E2 -20881.877} C_VEL
LIN {X 0,Y 214.195,Z 354.116,A -85,B 0,C 180,E1 -20888.728,E2 -20888.728} C_VEL
LIN {X 0,Y 215.476,Z 360.168,A -85,B 0,C 180,E1 -20894.159,E2 -20894.159} C_VEL
LIN {X 0,Y 216.924,Z 366.171,A -85,B 0,C 180,E1 -20898.903,E2 -20898.903} C_VEL
LIN {X 0,Y 218.289,Z 371.385,A -85,B 0,C 180,E1 -20902.727,E2 -20902.727} C_VEL
LIN {X 0,Y 220.074,Z 378.631,A -85,B 0,C 180,E1 -20907.583,E2 -20907.583} C_VEL
LIN {X 0,Y 221.803,Z 385.106,A -85,B 0,C 180,E1 -20911.608,E2 -20911.608} C_VEL
LIN {X 0,Y 223.698,Z 392.165,A -85,B 0,C 180,E1 -20915.686,E2 -20915.686} C_VEL
LIN {X 0,Y 226.235,Z 401.623,A -85,B 0,C 180,E1 -20920.719,E2 -20920.719} C_VEL
LIN {X 0,Y 228.045,Z 408.233,A -85,B 0,C 180,E1 -20923.977,E2 -20923.977} C_VEL
LIN {X 0,Y 233.264,Z 421.688,A -85,B 0,C 180,E1 -20925.38,E2 -20925.38} C_VEL
LIN {X 0,Y 234.246,Z 435.609,A -85,B 0,C 180,E1 -20926.46,E2 -20926.46} C_VEL
LIN {X 0,Y 234.104,Z 441.31,A -85,B 0,C 180,E1 -20926.918,E2 -20926.918} C_VEL
LIN {X 0,Y 231.951,Z 450.698,A -85,B 0,C 180,E1 -20927.597,E2 -20927.597} C_VEL
LIN {X 0,Y 229.651,Z 459.74,A -85,B 0,C 180,E1 -20928.369,E2 -20928.369} C_VEL
LIN {X 0,Y 229.242,Z 465.006,A -85,B 0,C 180,E1 -20928.968,E2 -20928.968} C_VEL
LIN {X 0,Y 229.594,Z 476.981,A -85,B 0,C 180,E1 -20930.574,E2 -20930.574} C_VEL
LIN {X 0,Y 226.288,Z 490.672,A -85,B 0,C 180,E1 -20932.453,E2 -20932.453} C_VEL
LIN {X 0,Y 222.612,Z 504.761,A -85,B 0,C 180,E1 -20934.825,E2 -20934.825} C_VEL
LIN {X 0,Y 218.919,Z 517.678,A -85,B 0,C 180,E1 -20937.477,E2 -20937.477} C_VEL
LIN {X 0,Y 215.292,Z 530.442,A -85,B 0,C 180,E1 -20940.688,E2 -20940.688} C_VEL
LIN {X 0,Y 212.245,Z 541.384,A -85,B 0,C 180,E1 -20944.05,E2 -20944.05} C_VEL
LIN {X 0,Y 209.697,Z 551.501,A -85,B 0,C 180,E1 -20947.855,E2 -20947.855} C_VEL
LIN {X 0,Y 208.023,Z 559.949,A -85,B 0,C 180,E1 -20951.766,E2 -20951.766} C_VEL
LIN {X 0,Y 206.771,Z 568.158,A -85,B 0,C 180,E1 -20956.241,E2 -20956.241} C_VEL
LIN {X 0,Y 206.474,Z 572.476,A -85,B 0,C 180,E1 -20959.215,E2 -20959.215} C_VEL
LIN {X 0,Y 206.462,Z 575.695,A -85,B 0,C 180,E1 -20962.179,E2 -20962.179} C_VEL
LIN {X 0,Y 206.521,Z 577.257,A -85,B 0,C 180,E1 -20964.145,E2 -20964.145} C_VEL
LIN {X 0,Y 206.679,Z 578.374,A -85,B 0,C 180,E1 -20966.105,E2 -20966.105} C_VEL
LIN {X 0,Y 206.924,Z 579.847,A -85,B 0,C 180,E1 -20970.005,E2 -20970.005} C_VEL
LIN {X 0,Y 206.434,Z 580.274,A -85,B 0,C 180,E1 -20973.909,E2 -20973.909} C_VEL
LIN {X 0,Y 205.921,Z 579.623,A -85,B 0,C 180,E1 -20977.851,E2 -20977.851} C_VEL
LIN {X 0,Y 205.739,Z 577.884,A -85,B 0,C 180,E1 -20981.832,E2 -20981.832} C_VEL
LIN {X 0,Y 206.321,Z 575.295,A -85,B 0,C 180,E1 -20985.818,E2 -20985.818} C_VEL
LIN {X 0,Y 208.129,Z 570.745,A -85,B 0,C 180,E1 -20990.771,E2 -20990.771} C_VEL
LIN {X 0,Y 211.443,Z 564.898,A -85,B 0,C 180,E1 -20995.605,E2 -20995.605} C_VEL
LIN {X 0,Y 216.288,Z 557.781,A -85,B 0,C 180,E1 -21000.246,E2 -21000.246} C_VEL
LIN {X 0,Y 222.748,Z 549.427,A -85,B 0,C 180,E1 -21004.61,E2 -21004.61} C_VEL
LIN {X 0,Y 231.624,Z 538.753,A -85,B 0,C 180,E1 -21009.025,E2 -21009.025} C_VEL
LIN {X 0,Y 241.232,Z 527.661,A -85,B 0,C 180,E1 -21012.642,E2 -21012.642} C_VEL
LIN {X 0,Y 249.702,Z 518.001,A -85,B 0,C 180,E1 -21015.179,E2 -21015.179} C_VEL
LIN {X 0,Y 259.43,Z 506.788,A -85,B 0,C 180,E1 -21017.583,E2 -21017.583} C_VEL
LIN {X 0,Y 266.858,Z 498.011,A -85,B 0,C 180,E1 -21019.219,E2 -21019.219} C_VEL
LIN {X 0,Y 272.624,Z 490.781,A -85,B 0,C 180,E1 -21020.662,E2 -21020.662} C_VEL
LIN {X 0,Y 272.46,Z 490.211,A -85,B 0,C 180,E1 -21021.753,E2 -21021.753} C_VEL
LIN {X 0,Y 271.509,Z 490.826,A -85,B 0,C 180,E1 -21022.534,E2 -21022.534} C_VEL
LIN {X 0,Y 262.022,Z 499.422,A -85,B 0,C 180,E1 -21024.784,E2 -21024.784} C_VEL
LIN {X 0,Y 253.225,Z 506.759,A -85,B 0,C 180,E1 -21027.235,E2 -21027.235} C_VEL
LIN {X 0,Y 245.182,Z 512.884,A -85,B 0,C 180,E1 -21029.893,E2 -21029.893} C_VEL
LIN {X 0,Y 237.849,Z 517.926,A -85,B 0,C 180,E1 -21032.743,E2 -21032.743} C_VEL
LIN {X 0,Y 232.909,Z 520.991,A -85,B 0,C 180,E1 -21035.012,E2 -21035.012} C_VEL
LIN {X 0,Y 226.952,Z 524.088,A -85,B 0,C 180,E1 -21038.186,E2 -21038.186} C_VEL
LIN {X 0,Y 221.768,Z 526.053,A -85,B 0,C 180,E1 -21041.525,E2 -21041.525} C_VEL
LIN {X 0,Y 217.434,Z 526.816,A -85,B 0,C 180,E1 -21045.015,E2 -21045.015} C_VEL
LIN {X 0,Y 214.042,Z 526.31,A -85,B 0,C 180,E1 -21048.639,E2 -21048.639} C_VEL
LIN {X 0,Y 211.354,Z 524.512,A -85,B 0,C 180,E1 -21052.357,E2 -21052.357} C_VEL
LIN {X 0,Y 210.395,Z 523.078,A -85,B 0,C 180,E1 -21054.249,E2 -21054.249} C_VEL
LIN {X 0,Y 209.038,Z 520.308,A -85,B 0,C 180,E1 -21057.11,E2 -21057.11} C_VEL
LIN {X 0,Y 208.009,Z 515.225,A -85,B 0,C 180,E1 -21060.969,E2 -21060.969} C_VEL
LIN {X 0,Y 207.779,Z 508.518,A -85,B 0,C 180,E1 -21064.852,E2 -21064.852} C_VEL
LIN {X 0,Y 207.929,Z 501.181,A -85,B 0,C 180,E1 -21068.26,E2 -21068.26} C_VEL
LIN {X 0,Y 208.872,Z 492.229,A -85,B 0,C 180,E1 -21071.648,E2 -21071.648} C_VEL
LIN {X 0,Y 209.994,Z 481.462,A -85,B 0,C 180,E1 -21075.034,E2 -21075.034} C_VEL
LIN {X 0,Y 211.609,Z 469.431,A -85,B 0,C 180,E1 -21078.142,E2 -21078.142} C_VEL
LIN {X 0,Y 213.517,Z 456.152,A -85,B 0,C 180,E1 -21080.975,E2 -21080.975} C_VEL
LIN {X 0,Y 215.533,Z 442.171,A -85,B 0,C 180,E1 -21083.448,E2 -21083.448} C_VEL
LIN {X 0,Y 217.379,Z 427.324,A -85,B 0,C 180,E1 -21085.622,E2 -21085.622} C_VEL
LIN {X 0,Y 217.76,Z 422.749,A -85,B 0,C 180,E1 -21086.216,E2 -21086.216} C_VEL
LIN {X 0,Y 215.284,Z 408.589,A -85,B 0,C 180,E1 -21088.178,E2 -21088.178} C_VEL
LIN {X 0,Y 211.623,Z 391.715,A -85,B 0,C 180,E1 -21090.222,E2 -21090.222} C_VEL
LIN {X 0,Y 208.828,Z 379.651,A -85,B 0,C 180,E1 -21091.546,E2 -21091.546} C_VEL
LIN {X 0,Y 209.202,Z 377.265,A -85,B 0,C 180,E1 -21093.603,E2 -21093.603} C_VEL
LIN {X 0,Y 212.869,Z 380.93,A -85,B 0,C 180,E1 -21097.586,E2 -21097.586} C_VEL
LIN {X 0,Y 214.357,Z 383.282,A -85,B 0,C 180,E1 -21099.743,E2 -21099.743} C_VEL
LIN {X 0,Y 215.571,Z 386.079,A -85,B 0,C 180,E1 -21101.939,E2 -21101.939} C_VEL
LIN {X 0,Y 216.393,Z 389.625,A -85,B 0,C 180,E1 -21104.391,E2 -21104.391} C_VEL
LIN {X 0,Y 217.387,Z 396.155,A -85,B 0,C 180,E1 -21108.617,E2 -21108.617} C_VEL
LIN {X 0,Y 217.68,Z 399.83,A -85,B 0,C 180,E1 -21110.794,E2 -21110.794} C_VEL
LIN {X 0,Y 217.126,Z 408.403,A -85,B 0,C 180,E1 -21115.248,E2 -21115.248} C_VEL
LIN {X 0,Y 222.552,Z 422.154,A -85,B 0,C 180,E1 -21117.017,E2 -21117.017} C_VEL
LIN {X 0,Y 225.713,Z 432.018,A -85,B 0,C 180,E1 -21118.428,E2 -21118.428} C_VEL
LIN {X 0,Y 227.474,Z 439.435,A -85,B 0,C 180,E1 -21119.564,E2 -21119.564} C_VEL
LIN {X 0,Y 227.104,Z 443.723,A -85,B 0,C 180,E1 -21120.055,E2 -21120.055} C_VEL
LIN {X 0,Y 225.095,Z 456.084,A -85,B 0,C 180,E1 -21121.658,E2 -21121.658} C_VEL
LIN {X 0,Y 222.808,Z 467.154,A -85,B 0,C 180,E1 -21123.538,E2 -21123.538} C_VEL
LIN {X 0,Y 220.54,Z 476.453,A -85,B 0,C 180,E1 -21125.522,E2 -21125.522} C_VEL
LIN {X 0,Y 218.247,Z 484.921,A -85,B 0,C 180,E1 -21127.763,E2 -21127.763} C_VEL
LIN {X 0,Y 215.748,Z 493.15,A -85,B 0,C 180,E1 -21130.49,E2 -21130.49} C_VEL
LIN {X 0,Y 213.386,Z 500.652,A -85,B 0,C 180,E1 -21133.738,E2 -21133.738} C_VEL
LIN {X 0,Y 211.408,Z 505.72,A -85,B 0,C 180,E1 -21136.539,E2 -21136.539} C_VEL
LIN {X 0,Y 209.902,Z 509.624,A -85,B 0,C 180,E1 -21139.384,E2 -21139.384} C_VEL
LIN {X 0,Y 209.041,Z 512.456,A -85,B 0,C 180,E1 -21142.267,E2 -21142.267} C_VEL
LIN {X 0,Y 208.574,Z 513.833,A -85,B 0,C 180,E1 -21144.194,E2 -21144.194} C_VEL
LIN {X 0,Y 208.031,Z 515.395,A -85,B 0,C 180,E1 -21148.059,E2 -21148.059} C_VEL
LIN {X 0,Y 207.946,Z 515.624,A -85,B 0,C 180,E1 -21149.995,E2 -21149.995} C_VEL
LIN {X 0,Y 208.243,Z 514.854,A -85,B 0,C 180,E1 -21153.866,E2 -21153.866} C_VEL
LIN {X 0,Y 208.59,Z 513.908,A -85,B 0,C 180,E1 -21155.796,E2 -21155.796} C_VEL
LIN {X 0,Y 209.034,Z 512.579,A -85,B 0,C 180,E1 -21157.724,E2 -21157.724} C_VEL
LIN {X 0,Y 209.877,Z 509.795,A -85,B 0,C 180,E1 -21160.608,E2 -21160.608} C_VEL
LIN {X 0,Y 211.383,Z 505.946,A -85,B 0,C 180,E1 -21163.453,E2 -21163.453} C_VEL
LIN {X 0,Y 213.347,Z 500.938,A -85,B 0,C 180,E1 -21166.255,E2 -21166.255} C_VEL
LIN {X 0,Y 215.314,Z 494.677,A -85,B 0,C 180,E1 -21169.046,E2 -21169.046} C_VEL
LIN {X 0,Y 217.74,Z 486.858,A -85,B 0,C 180,E1 -21171.783,E2 -21171.783} C_VEL
LIN {X 0,Y 220.045,Z 478.838,A -85,B 0,C 180,E1 -21174.025,E2 -21174.025} C_VEL
LIN {X 0,Y 221.933,Z 471.116,A -85,B 0,C 180,E1 -21175.807,E2 -21175.807} C_VEL
LIN {X 0,Y 224.273,Z 460.532,A -85,B 0,C 180,E1 -21177.778,E2 -21177.778} C_VEL
LIN {X 0,Y 226.3,Z 449.765,A -85,B 0,C 180,E1 -21179.339,E2 -21179.339} C_VEL
LIN {X 0,Y 227.65,Z 440.146,A -85,B 0,C 180,E1 -21180.462,E2 -21180.462} C_VEL
LIN {X 0,Y 224.686,Z 428.558,A -85,B 0,C 180,E1 -21182.22,E2 -21182.22} C_VEL
LIN {X 0,Y 220.801,Z 417.421,A -85,B 0,C 180,E1 -21183.759,E2 -21183.759} C_VEL
LIN {X 0,Y 217.208,Z 408.388,A -85,B 0,C 180,E1 -21184.901,E2 -21184.901} C_VEL
LIN {X 0,Y 217.667,Z 400.158,A -85,B 0,C 180,E1 -21189.202,E2 -21189.202} C_VEL
LIN {X 0,Y 217.256,Z 395.563,A -85,B 0,C 180,E1 -21191.923,E2 -21191.923} C_VEL
LIN {X 0,Y 216.322,Z 389.073,A -85,B 0,C 180,E1 -21196.17,E2 -21196.17} C_VEL
LIN {X 0,Y 215.269,Z 382.939,A -85,B 0,C 180,E1 -21200.458,E2 -21200.458} C_VEL
LIN {X 0,Y 214.274,Z 378.276,A -85,B 0,C 180,E1 -21203.815,E2 -21203.815} C_VEL
LIN {X 0,Y 212.918,Z 373.025,A -85,B 0,C 180,E1 -21208.12,E2 -21208.12} C_VEL
LIN {X 0,Y 211.809,Z 369.045,A -85,B 0,C 180,E1 -21211.24,E2 -21211.24} C_VEL
LIN {X 0,Y 210.692,Z 365.634,A -85,B 0,C 180,E1 -21214.301,E2 -21214.301} C_VEL
LIN {X 0,Y 209.328,Z 361.799,A -85,B 0,C 180,E1 -21218.326,E2 -21218.326} C_VEL
LIN {X 0,Y 208.587,Z 359.679,A -85,B 0,C 180,E1 -21220.615,E2 -21220.615} C_VEL
LIN {X 0,Y 206.876,Z 355.011,A -85,B 0,C 180,E1 -21225.615,E2 -21225.615} C_VEL
LIN {X 0,Y 207.085,Z 354.983,A -85,B 0,C 180,E1 -21230.23,E2 -21230.23} C_VEL
LIN {X 0,Y 207.157,Z 354.985,A -85,B 0,C 180,E1 -21232.2,E2 -21232.2} C_VEL
LIN {X 0,Y 207.359,Z 354.969,A -85,B 0,C 180,E1 -21238.057,E2 -21238.057} C_VEL
LIN {X 0,Y 207.49,Z 354.933,A -85,B 0,C 180,E1 -21239.999,E2 -21239.999} C_VEL
LIN {X 0,Y 207.395,Z 354.948,A -85,B 0,C 180,E1 -21241.941,E2 -21241.941} C_VEL
LIN {X 0,Y 207.175,Z 355.007,A -85,B 0,C 180,E1 -21247.308,E2 -21247.308} C_VEL
LIN {X 0,Y 208.143,Z 359.854,A -85,B 0,C 180,E1 -21251.738,E2 -21251.738} C_VEL
LIN {X 0,Y 209.537,Z 365.57,A -85,B 0,C 180,E1 -21256.564,E2 -21256.564} C_VEL
LIN {X 0,Y 211.122,Z 371.951,A -85,B 0,C 180,E1 -21261.479,E2 -21261.479} C_VEL
LIN {X 0,Y 212.532,Z 377.569,A -85,B 0,C 180,E1 -21265.459,E2 -21265.459} C_VEL
LIN {X 0,Y 214.557,Z 385.312,A -85,B 0,C 180,E1 -21270.511,E2 -21270.511} C_VEL
LIN {X 0,Y 216.947,Z 394.419,A -85,B 0,C 180,E1 -21275.926,E2 -21275.926} C_VEL
LIN {X 0,Y 219.477,Z 403.788,A -85,B 0,C 180,E1 -21281.028,E2 -21281.028} C_VEL
LIN {X 0,Y 220.57,Z 407.714,A -85,B 0,C 180,E1 -21283.047,E2 -21283.047} C_VEL
LIN {X 0,Y 226.834,Z 423.829,A -85,B 0,C 180,E1 -21284.805,E2 -21284.805} C_VEL
LIN {X 0,Y 227.854,Z 440.277,A -85,B 0,C 180,E1 -21286.215,E2 -21286.215} C_VEL
LIN {X 0,Y 228.778,Z 457.023,A -85,B 0,C 180,E1 -21287.989,E2 -21287.989} C_VEL
LIN {X 0,Y 229.242,Z 465.006,A -85,B 0,C 180,E1 -21288.968,E2 -21288.968} C_VEL
LIN {X 0,Y 229.005,Z 468.554,A -85,B 0,C 180,E1 -21289.389,E2 -21289.389} C_VEL
LIN {X 0,Y 228.118,Z 472.069,A -85,B 0,C 180,E1 -21289.779,E2 -21289.779} C_VEL
LIN {X 0,Y 225.147,Z 478.87,A -85,B 0,C 180,E1 -21290.517,E2 -21290.517} C_VEL
LIN {X 0,Y 220.111,Z 488.879,A -85,B 0,C 180,E1 -21291.765,E2 -21291.765} C_VEL
LIN {X 0,Y 218.982,Z 492.203,A -85,B 0,C 180,E1 -21292.281,E2 -21292.281} C_VEL
LIN {X 0,Y 215.38,Z 505.539,A -85,B 0,C 180,E1 -21294.662,E2 -21294.662} C_VEL
LIN {X 0,Y 211.717,Z 518.011,A -85,B 0,C 180,E1 -21297.362,E2 -21297.362} C_VEL
LIN {X 0,Y 208.524,Z 528.883,A -85,B 0,C 180,E1 -21300.196,E2 -21300.196} C_VEL
LIN {X 0,Y 205.462,Z 539.694,A -85,B 0,C 180,E1 -21303.603,E2 -21303.603} C_VEL
LIN {X 0,Y 202.786,Z 550.054,A -85,B 0,C 180,E1 -21307.596,E2 -21307.596} C_VEL
LIN {X 0,Y 200.608,Z 561.546,A -85,B 0,C 180,E1 -21312.681,E2 -21312.681} C_VEL
LIN {X 0,Y 199.777,Z 567.057,A -85,B 0,C 180,E1 -21315.749,E2 -21315.749} C_VEL
LIN {X 0,Y 199.415,Z 571.375,A -85,B 0,C 180,E1 -21318.828,E2 -21318.828} C_VEL
LIN {X 0,Y 199.399,Z 574.597,A -85,B 0,C 180,E1 -21321.9,E2 -21321.9} C_VEL
LIN {X 0,Y 199.46,Z 576.156,A -85,B 0,C 180,E1 -21323.937,E2 -21323.937} C_VEL
LIN {X 0,Y 199.622,Z 577.275,A -85,B 0,C 180,E1 -21325.967,E2 -21325.967} C_VEL
LIN {X 0,Y 199.845,Z 577.976,A -85,B 0,C 180,E1 -21327.99,E2 -21327.99} C_VEL
LIN {X 0,Y 199.996,Z 578.314,A -85,B 0,C 180,E1 -21330.005,E2 -21330.005} C_VEL
LIN {X 0,Y 199.466,Z 578.875,A -85,B 0,C 180,E1 -21334.046,E2 -21334.046} C_VEL
LIN {X 0,Y 198.889,Z 578.314,A -85,B 0,C 180,E1 -21338.13,E2 -21338.13} C_VEL
LIN {X 0,Y 198.739,Z 576.73,A -85,B 0,C 180,E1 -21342.255,E2 -21342.255} C_VEL
LIN {X 0,Y 199.391,Z 574.247,A -85,B 0,C 180,E1 -21346.383,E2 -21346.383} C_VEL
LIN {X 0,Y 200.846,Z 570.921,A -85,B 0,C 180,E1 -21350.487,E2 -21350.487} C_VEL
LIN {X 0,Y 204.064,Z 565.594,A -85,B 0,C 180,E1 -21355.504,E2 -21355.504} C_VEL
LIN {X 0,Y 208.91,Z 559.024,A -85,B 0,C 180,E1 -21360.311,E2 -21360.311} C_VEL
LIN {X 0,Y 215.423,Z 551.29,A -85,B 0,C 180,E1 -21364.819,E2 -21364.819} C_VEL
LIN {X 0,Y 223.45,Z 542.379,A -85,B 0,C 180,E1 -21368.984,E2 -21368.984} C_VEL
LIN {X 0,Y 233.012,Z 532.248,A -85,B 0,C 180,E1 -21372.742,E2 -21372.742} C_VEL
LIN {X 0,Y 241.536,Z 523.302,A -85,B 0,C 180,E1 -21375.414,E2 -21375.414} C_VEL
LIN {X 0,Y 253.646,Z 510.598,A -85,B 0,C 180,E1 -21378.432,E2 -21378.432} C_VEL
LIN {X 0,Y 262.651,Z 500.965,A -85,B 0,C 180,E1 -21380.295,E2 -21380.295} C_VEL
LIN {X 0,Y 266.204,Z 496.889,A -85,B 0,C 180,E1 -21381.157,E2 -21381.157} C_VEL
LIN {X 0,Y 267.469,Z 495.373,A -85,B 0,C 180,E1 -21381.598,E2 -21381.598} C_VEL
LIN {X 0,Y 257.059,Z 503.856,A -85,B 0,C 180,E1 -21383.999,E2 -21383.999} C_VEL
LIN {X 0,Y 245.806,Z 512.189,A -85,B 0,C 180,E1 -21387.096,E2 -21387.096} C_VEL
LIN {X 0,Y 235.786,Z 518.695,A -85,B 0,C 180,E1 -21390.541,E2 -21390.541} C_VEL
LIN {X 0,Y 230.3,Z 521.863,A -85,B 0,C 180,E1 -21392.759,E2 -21392.759} C_VEL
LIN {X 0,Y 223.723,Z 525.115,A -85,B 0,C 180,E1 -21395.898,E2 -21395.898} C_VEL
LIN {X 0,Y 217.919,Z 527.299,A -85,B 0,C 180,E1 -21399.222,E2 -21399.222} C_VEL
LIN {X 0,Y 212.91,Z 528.355,A -85,B 0,C 180,E1 -21402.718,E2 -21402.718} C_VEL
LIN {X 0,Y 208.84,Z 528.194,A -85,B 0,C 180,E1 -21406.376,E2 -21406.376} C_VEL
LIN {X 0,Y 205.742,Z 526.756,A -85,B 0,C 180,E1 -21410.167,E2 -21410.167} C_VEL
LIN {X 0,Y 203.394,Z 523.998,A -85,B 0,C 180,E1 -21414.051,E2 -21414.051} C_VEL
LIN {X 0,Y 201.993,Z 520.997,A -85,B 0,C 180,E1 -21417.009,E2 -21417.009} C_VEL
LIN {X 0,Y 200.939,Z 515.672,A -85,B 0,C 180,E1 -21421.003,E2 -21421.003} C_VEL
LIN {X 0,Y 200.694,Z 510.601,A -85,B 0,C 180,E1 -21424.017,E2 -21424.017} C_VEL
LIN {X 0,Y 200.816,Z 502.301,A -85,B 0,C 180,E1 -21428.048,E2 -21428.048} C_VEL
LIN {X 0,Y 201.752,Z 493.363,A -85,B 0,C 180,E1 -21431.555,E2 -21431.555} C_VEL
LIN {X 0,Y 202.873,Z 482.544,A -85,B 0,C 180,E1 -21435.06,E2 -21435.06} C_VEL
LIN {X 0,Y 204.53,Z 470.597,A -85,B 0,C 180,E1 -21438.274,E2 -21438.274} C_VEL
LIN {X 0,Y 206.196,Z 458.548,A -85,B 0,C 180,E1 -21440.971,E2 -21440.971} C_VEL
LIN {X 0,Y 208.154,Z 445.701,A -85,B 0,C 180,E1 -21443.374,E2 -21443.374} C_VEL
LIN {X 0,Y 210.016,Z 432.207,A -85,B 0,C 180,E1 -21445.501,E2 -21445.501} C_VEL
LIN {X 0,Y 210.902,Z 425.128,A -85,B 0,C 180,E1 -21446.469,E2 -21446.469} C_VEL
LIN {X 0,Y 209.531,Z 415.824,A -85,B 0,C 180,E1 -21447.835,E2 -21447.835} C_VEL
LIN {X 0,Y 206.39,Z 399.817,A -85,B 0,C 180,E1 -21449.973,E2 -21449.973} C_VEL
LIN {X 0,Y 202.481,Z 382.423,A -85,B 0,C 180,E1 -21451.994,E2 -21451.994} C_VEL
LIN {X 0,Y 201.954,Z 380.255,A -85,B 0,C 180,E1 -21452.244,E2 -21452.244} C_VEL
LIN {X 0,Y 205.096,Z 382.955,A -85,B 0,C 180,E1 -21455.63,E2 -21455.63} C_VEL
LIN {X 0,Y 206.936,Z 384.782,A -85,B 0,C 180,E1 -21457.686,E2 -21457.686} C_VEL
LIN {X 0,Y 208.987,Z 388.468,A -85,B 0,C 180,E1 -21460.979,E2 -21460.979} C_VEL
LIN {X 0,Y 209.888,Z 391.599,A -85,B 0,C 180,E1 -21463.348,E2 -21463.348} C_VEL
LIN {X 0,Y 210.82,Z 397.364,A -85,B 0,C 180,E1 -21467.173,E2 -21467.173} C_VEL
LIN {X 0,Y 211.285,Z 401.733,A -85,B 0,C 180,E1 -21469.913,E2 -21469.913} C_VEL
LIN {X 0,Y 210.831,Z 409.675,A -85,B 0,C 180,E1 -21474.089,E2 -21474.089} C_VEL
LIN {X 0,Y 216.04,Z 422.699,A -85,B 0,C 180,E1 -21475.846,E2 -21475.846} C_VEL
LIN {X 0,Y 219.542,Z 433.688,A -85,B 0,C 180,E1 -21477.496,E2 -21477.496} C_VEL
LIN {X 0,Y 221.264,Z 441.006,A -85,B 0,C 180,E1 -21478.676,E2 -21478.676} C_VEL
LIN {X 0,Y 221.09,Z 444.581,A -85,B 0,C 180,E1 -21479.125,E2 -21479.125} C_VEL
LIN {X 0,Y 219.183,Z 455.903,A -85,B 0,C 180,E1 -21480.605,E2 -21480.605} C_VEL
LIN {X 0,Y 216.831,Z 467.094,A -85,B 0,C 180,E1 -21482.487,E2 -21482.487} C_VEL
LIN {X 0,Y 214.621,Z 475.66,A -85,B 0,C 180,E1 -21484.281,E2 -21484.281} C_VEL
LIN {X 0,Y 212.722,Z 482.824,A -85,B 0,C 180,E1 -21486.122,E2 -21486.122} C_VEL
LIN {X 0,Y 209.976,Z 491.673,A -85,B 0,C 180,E1 -21488.907,E2 -21488.907} C_VEL
LIN {X 0,Y 207.82,Z 498.344,A -85,B 0,C 180,E1 -21491.578,E2 -21491.578} C_VEL
LIN {X 0,Y 205.972,Z 503.533,A -85,B 0,C 180,E1 -21494.154,E2 -21494.154} C_VEL
LIN {X 0,Y 204.043,Z 508.196,A -85,B 0,C 180,E1 -21497.058,E2 -21497.058} C_VEL
LIN {X 0,Y 202.683,Z 511.731,A -85,B 0,C 180,E1 -21500.011,E2 -21500.011} C_VEL
LIN {X 0,Y 202.089,Z 513.533,A -85,B 0,C 180,E1 -21501.999,E2 -21501.999} C_VEL
LIN {X 0,Y 201.605,Z 514.909,A -85,B 0,C 180,E1 -21503.992,E2 -21503.992} C_VEL
LIN {X 0,Y 201.02,Z 516.472,A -85,B 0,C 180,E1 -21507.992,E2 -21507.992} C_VEL
LIN {X 0,Y 200.929,Z 516.701,A -85,B 0,C 180,E1 -21509.995,E2 -21509.995} C_VEL
LIN {X 0,Y 201.256,Z 515.928,A -85,B 0,C 180,E1 -21514,E2 -21514} C_VEL
LIN {X 0,Y 201.619,Z 514.983,A -85,B 0,C 180,E1 -21515.998,E2 -21515.998} C_VEL
LIN {X 0,Y 202.081,Z 513.655,A -85,B 0,C 180,E1 -21517.991,E2 -21517.991} C_VEL
LIN {X 0,Y 202.981,Z 510.871,A -85,B 0,C 180,E1 -21520.973,E2 -21520.973} C_VEL
LIN {X 0,Y 204.565,Z 507.021,A -85,B 0,C 180,E1 -21523.91,E2 -21523.91} C_VEL
LIN {X 0,Y 206.625,Z 502.01,A -85,B 0,C 180,E1 -21526.8,E2 -21526.8} C_VEL
LIN {X 0,Y 209.108,Z 494.564,A -85,B 0,C 180,E1 -21530.146,E2 -21530.146} C_VEL
LIN {X 0,Y 211.645,Z 486.465,A -85,B 0,C 180,E1 -21532.96,E2 -21532.96} C_VEL
LIN {X 0,Y 213.651,Z 479.905,A -85,B 0,C 180,E1 -21534.792,E2 -21534.792} C_VEL
LIN {X 0,Y 215.634,Z 472.18,A -85,B 0,C 180,E1 -21536.619,E2 -21536.619} C_VEL
LIN {X 0,Y 218.086,Z 461.59,A -85,B 0,C 180,E1 -21538.638,E2 -21538.638} C_VEL
LIN {X 0,Y 220.224,Z 450.773,A -85,B 0,C 180,E1 -21540.238,E2 -21540.238} C_VEL
LIN {X 0,Y 221.547,Z 442.104,A -85,B 0,C 180,E1 -21541.28,E2 -21541.28} C_VEL
LIN {X 0,Y 218.654,Z 430.435,A -85,B 0,C 180,E1 -21543.14,E2 -21543.14} C_VEL
LIN {X 0,Y 214.513,Z 418.335,A -85,B 0,C 180,E1 -21544.898,E2 -21544.898} C_VEL
LIN {X 0,Y 210.846,Z 409.541,A -85,B 0,C 180,E1 -21546.069,E2 -21546.069} C_VEL
LIN {X 0,Y 211.28,Z 403.627,A -85,B 0,C 180,E1 -21549.192,E2 -21549.192} C_VEL
LIN {X 0,Y 211.06,Z 399.342,A -85,B 0,C 180,E1 -21551.75,E2 -21551.75} C_VEL
LIN {X 0,Y 210.044,Z 391.903,A -85,B 0,C 180,E1 -21556.692,E2 -21556.692} C_VEL
LIN {X 0,Y 208.903,Z 385.38,A -85,B 0,C 180,E1 -21561.345,E2 -21561.345} C_VEL
LIN {X 0,Y 207.892,Z 380.689,A -85,B 0,C 180,E1 -21564.92,E2 -21564.92} C_VEL
LIN {X 0,Y 206.621,Z 375.431,A -85,B 0,C 180,E1 -21569.321,E2 -21569.321} C_VEL
LIN {X 0,Y 205.383,Z 370.832,A -85,B 0,C 180,E1 -21573.586,E2 -21573.586} C_VEL
LIN {X 0,Y 203.76,Z 366.569,A -85,B 0,C 180,E1 -21577.702,E2 -21577.702} C_VEL
LIN {X 0,Y 202.71,Z 363.079,A -85,B 0,C 180,E1 -21581.817,E2 -21581.817} C_VEL
LIN {X 0,Y 201.404,Z 359.528,A -85,B 0,C 180,E1 -21585.861,E2 -21585.861} C_VEL
LIN {X 0,Y 200.181,Z 356.572,A -85,B 0,C 180,E1 -21590.909,E2 -21590.909} C_VEL
LIN {X 0,Y 200.099,Z 355.86,A -85,B 0,C 180,E1 -21591.923,E2 -21591.923} C_VEL
LIN {X 0,Y 200.299,Z 355.849,A -85,B 0,C 180,E1 -21597.988,E2 -21597.988} C_VEL
LIN {X 0,Y 200.455,Z 355.809,A -85,B 0,C 180,E1 -21599.999,E2 -21599.999} C_VEL
LIN {X 0,Y 200.331,Z 355.828,A -85,B 0,C 180,E1 -21602.01,E2 -21602.01} C_VEL
LIN {X 0,Y 200.023,Z 355.99,A -85,B 0,C 180,E1 -21605.67,E2 -21605.67} C_VEL
LIN {X 0,Y 200.941,Z 359.386,A -85,B 0,C 180,E1 -21609.055,E2 -21609.055} C_VEL
LIN {X 0,Y 202.423,Z 366.181,A -85,B 0,C 180,E1 -21615.093,E2 -21615.093} C_VEL
LIN {X 0,Y 203.96,Z 372.464,A -85,B 0,C 180,E1 -21620.155,E2 -21620.155} C_VEL
LIN {X 0,Y 205.338,Z 377.994,A -85,B 0,C 180,E1 -21624.249,E2 -21624.249} C_VEL
LIN {X 0,Y 207.294,Z 385.629,A -85,B 0,C 180,E1 -21629.445,E2 -21629.445} C_VEL
LIN {X 0,Y 209.072,Z 392.379,A -85,B 0,C 180,E1 -21633.686,E2 -21633.686} C_VEL
LIN {X 0,Y 211.036,Z 399.823,A -85,B 0,C 180,E1 -21638.031,E2 -21638.031} C_VEL
LIN {X 0,Y 213.156,Z 407.379,A -85,B 0,C 180,E1 -21642.125,E2 -21642.125} C_VEL
LIN {X 0,Y 220.355,Z 426.026,A -85,B 0,C 180,E1 -21644.24,E2 -21644.24} C_VEL
LIN {X 0,Y 221.286,Z 442.648,A -85,B 0,C 180,E1 -21645.767,E2 -21645.767} C_VEL
LIN {X 0,Y 222.122,Z 459.167,A -85,B 0,C 180,E1 -21647.634,E2 -21647.634} C_VEL
LIN {X 0,Y 222.683,Z 473.559,A -85,B 0,C 180,E1 -21649.565,E2 -21649.565} C_VEL
LIN {X 0,Y 222.73,Z 477.127,A -85,B 0,C 180,E1 -21650.091,E2 -21650.091} C_VEL
LIN {X 0,Y 219.149,Z 491.561,A -85,B 0,C 180,E1 -21652.176,E2 -21652.176} C_VEL
LIN {X 0,Y 218.982,Z 492.203,A -85,B 0,C 180,E1 -21652.281,E2 -21652.281} C_VEL
LIN {X 0,Y 217.047,Z 497.042,A -85,B 0,C 180,E1 -21653.045,E2 -21653.045} C_VEL
LIN {X 0,Y 207.98,Z 509.981,A -85,B 0,C 180,E1 -21655.334,E2 -21655.334} C_VEL
LIN {X 0,Y 205.711,Z 514.224,A -85,B 0,C 180,E1 -21656.271,E2 -21656.271} C_VEL
LIN {X 0,Y 205.233,Z 515.676,A -85,B 0,C 180,E1 -21656.613,E2 -21656.613} C_VEL
LIN {X 0,Y 201.814,Z 527.202,A -85,B 0,C 180,E1 -21659.678,E2 -21659.678} C_VEL
LIN {X 0,Y 198.656,Z 538.102,A -85,B 0,C 180,E1 -21663.194,E2 -21663.194} C_VEL
LIN {X 0,Y 196.415,Z 546.551,A -85,B 0,C 180,E1 -21666.269,E2 -21666.269} C_VEL
LIN {X 0,Y 194.623,Z 555.393,A -85,B 0,C 180,E1 -21669.662,E2 -21669.662} C_VEL
LIN {X 0,Y 193.352,Z 562.396,A -85,B 0,C 180,E1 -21673.101,E2 -21673.101} C_VEL
LIN {X 0,Y 192.601,Z 567.497,A -85,B 0,C 180,E1 -21676.285,E2 -21676.285} C_VEL
LIN {X 0,Y 192.357,Z 571.45,A -85,B 0,C 180,E1 -21679.479,E2 -21679.479} C_VEL
LIN {X 0,Y 192.342,Z 573.504,A -85,B 0,C 180,E1 -21681.601,E2 -21681.601} C_VEL
LIN {X 0,Y 192.402,Z 575.066,A -85,B 0,C 180,E1 -21683.714,E2 -21683.714} C_VEL
LIN {X 0,Y 192.562,Z 576.187,A -85,B 0,C 180,E1 -21685.819,E2 -21685.819} C_VEL
LIN {X 0,Y 192.799,Z 576.89,A -85,B 0,C 180,E1 -21687.916,E2 -21687.916} C_VEL
LIN {X 0,Y 192.993,Z 577.154,A -85,B 0,C 180,E1 -21690.005,E2 -21690.005} C_VEL
LIN {X 0,Y 192.485,Z 577.45,A -85,B 0,C 180,E1 -21694.193,E2 -21694.193} C_VEL
LIN {X 0,Y 191.853,Z 576.945,A -85,B 0,C 180,E1 -21698.484,E2 -21698.484} C_VEL
LIN {X 0,Y 191.736,Z 575.546,A -85,B 0,C 180,E1 -21702.71,E2 -21702.71} C_VEL
LIN {X 0,Y 193.126,Z 571.739,A -85,B 0,C 180,E1 -21709.123,E2 -21709.123} C_VEL
LIN {X 0,Y 196.71,Z 566.095,A -85,B 0,C 180,E1 -21715.392,E2 -21715.392} C_VEL
LIN {X 0,Y 201.547,Z 560.092,A -85,B 0,C 180,E1 -21720.377,E2 -21720.377} C_VEL
LIN {X 0,Y 208.092,Z 552.941,A -85,B 0,C 180,E1 -21725.045,E2 -21725.045} C_VEL
LIN {X 0,Y 216.18,Z 544.697,A -85,B 0,C 180,E1 -21729.347,E2 -21729.347} C_VEL
LIN {X 0,Y 225.814,Z 535.344,A -85,B 0,C 180,E1 -21733.217,E2 -21733.217} C_VEL
LIN {X 0,Y 234.461,Z 527,A -85,B 0,C 180,E1 -21736.01,E2 -21736.01} C_VEL
LIN {X 0,Y 247.87,Z 514.202,A -85,B 0,C 180,E1 -21739.321,E2 -21739.321} C_VEL
LIN {X 0,Y 257.169,Z 505.167,A -85,B 0,C 180,E1 -21741.161,E2 -21741.161} C_VEL
LIN {X 0,Y 258.133,Z 503.899,A -85,B 0,C 180,E1 -21741.8,E2 -21741.8} C_VEL
LIN {X 0,Y 247.347,Z 511.479,A -85,B 0,C 180,E1 -21744.376,E2 -21744.376} C_VEL
LIN {X 0,Y 238.379,Z 517.178,A -85,B 0,C 180,E1 -21746.947,E2 -21746.947} C_VEL
LIN {X 0,Y 228.19,Z 522.833,A -85,B 0,C 180,E1 -21750.477,E2 -21750.477} C_VEL
LIN {X 0,Y 220.949,Z 526.225,A -85,B 0,C 180,E1 -21753.557,E2 -21753.557} C_VEL
LIN {X 0,Y 214.505,Z 528.591,A -85,B 0,C 180,E1 -21756.849,E2 -21756.849} C_VEL
LIN {X 0,Y 208.858,Z 529.884,A -85,B 0,C 180,E1 -21760.337,E2 -21760.337} C_VEL
LIN {X 0,Y 204.126,Z 530.02,A -85,B 0,C 180,E1 -21764.013,E2 -21764.013} C_VEL
LIN {X 0,Y 200.403,Z 528.927,A -85,B 0,C 180,E1 -21767.854,E2 -21767.854} C_VEL
LIN {X 0,Y 197.441,Z 526.562,A -85,B 0,C 180,E1 -21771.815,E2 -21771.815} C_VEL
LIN {X 0,Y 195.808,Z 523.863,A -85,B 0,C 180,E1 -21774.853,E2 -21774.853} C_VEL
LIN {X 0,Y 194.301,Z 519.054,A -85,B 0,C 180,E1 -21778.965,E2 -21778.965} C_VEL
LIN {X 0,Y 193.661,Z 512.639,A -85,B 0,C 180,E1 -21783.121,E2 -21783.121} C_VEL
LIN {X 0,Y 193.623,Z 505.633,A -85,B 0,C 180,E1 -21786.776,E2 -21786.776} C_VEL
LIN {X 0,Y 194.235,Z 497.117,A -85,B 0,C 180,E1 -21790.424,E2 -21790.424} C_VEL
LIN {X 0,Y 195.211,Z 488.414,A -85,B 0,C 180,E1 -21793.56,E2 -21793.56} C_VEL
LIN {X 0,Y 196.481,Z 478.333,A -85,B 0,C 180,E1 -21796.629,E2 -21796.629} C_VEL
LIN {X 0,Y 198.382,Z 465.317,A -85,B 0,C 180,E1 -21799.938,E2 -21799.938} C_VEL
LIN {X 0,Y 200.401,Z 452.277,A -85,B 0,C 180,E1 -21802.692,E2 -21802.692} C_VEL
LIN {X 0,Y 202.281,Z 439.584,A -85,B 0,C 180,E1 -21804.938,E2 -21804.938} C_VEL
LIN {X 0,Y 204.024,Z 424.878,A -85,B 0,C 180,E1 -21807.112,E2 -21807.112} C_VEL
LIN {X 0,Y 201.237,Z 408.975,A -85,B 0,C 180,E1 -21809.49,E2 -21809.49} C_VEL
LIN {X 0,Y 197.472,Z 390.947,A -85,B 0,C 180,E1 -21811.828,E2 -21811.828} C_VEL
LIN {X 0,Y 196.096,Z 384.779,A -85,B 0,C 180,E1 -21812.579,E2 -21812.579} C_VEL
LIN {X 0,Y 196.996,Z 385.058,A -85,B 0,C 180,E1 -21813.277,E2 -21813.277} C_VEL
LIN {X 0,Y 199.999,Z 387.713,A -85,B 0,C 180,E1 -21816.684,E2 -21816.684} C_VEL
LIN {X 0,Y 200.984,Z 388.625,A -85,B 0,C 180,E1 -21817.731,E2 -21817.731} C_VEL
LIN {X 0,Y 202.978,Z 392.365,A -85,B 0,C 180,E1 -21821.138,E2 -21821.138} C_VEL
LIN {X 0,Y 203.789,Z 395.658,A -85,B 0,C 180,E1 -21823.61,E2 -21823.61} C_VEL
LIN {X 0,Y 204.78,Z 402.532,A -85,B 0,C 180,E1 -21828.201,E2 -21828.201} C_VEL
LIN {X 0,Y 204.853,Z 406.508,A -85,B 0,C 180,E1 -21830.598,E2 -21830.598} C_VEL
LIN {X 0,Y 204.591,Z 410.681,A -85,B 0,C 180,E1 -21832.81,E2 -21832.81} C_VEL
LIN {X 0,Y 209.612,Z 423.279,A -85,B 0,C 180,E1 -21834.606,E2 -21834.606} C_VEL
LIN {X 0,Y 212.851,Z 433.232,A -85,B 0,C 180,E1 -21836.166,E2 -21836.166} C_VEL
LIN {X 0,Y 215.149,Z 442.6,A -85,B 0,C 180,E1 -21837.747,E2 -21837.747} C_VEL
LIN {X 0,Y 215.321,Z 443.981,A -85,B 0,C 180,E1 -21837.964,E2 -21837.964} C_VEL
LIN {X 0,Y 213.303,Z 455.905,A -85,B 0,C 180,E1 -21839.519,E2 -21839.519} C_VEL
LIN {X 0,Y 211.214,Z 465.712,A -85,B 0,C 180,E1 -21841.148,E2 -21841.148} C_VEL
LIN {X 0,Y 208.561,Z 475.735,A -85,B 0,C 180,E1 -21843.206,E2 -21843.206} C_VEL
LIN {X 0,Y 206.348,Z 483.893,A -85,B 0,C 180,E1 -21845.336,E2 -21845.336} C_VEL
LIN {X 0,Y 203.444,Z 492.748,A -85,B 0,C 180,E1 -21848.196,E2 -21848.196} C_VEL
LIN {X 0,Y 201.212,Z 499.331,A -85,B 0,C 180,E1 -21850.906,E2 -21850.906} C_VEL
LIN {X 0,Y 199.231,Z 504.61,A -85,B 0,C 180,E1 -21853.603,E2 -21853.603} C_VEL
LIN {X 0,Y 197.209,Z 509.273,A -85,B 0,C 180,E1 -21856.601,E2 -21856.601} C_VEL
LIN {X 0,Y 195.777,Z 512.809,A -85,B 0,C 180,E1 -21859.655,E2 -21859.655} C_VEL
LIN {X 0,Y 195.14,Z 514.611,A -85,B 0,C 180,E1 -21861.712,E2 -21861.712} C_VEL
LIN {X 0,Y 194.636,Z 515.985,A -85,B 0,C 180,E1 -21863.776,E2 -21863.776} C_VEL
LIN {X 0,Y 194.009,Z 517.549,A -85,B 0,C 180,E1 -21867.919,E2 -21867.919} C_VEL
LIN {X 0,Y 193.911,Z 517.778,A -85,B 0,C 180,E1 -21869.995,E2 -21869.995} C_VEL
LIN {X 0,Y 194.267,Z 517.003,A -85,B 0,C 180,E1 -21874.144,E2 -21874.144} C_VEL
LIN {X 0,Y 194.647,Z 516.058,A -85,B 0,C 180,E1 -21876.213,E2 -21876.213} C_VEL
LIN {X 0,Y 195.133,Z 514.731,A -85,B 0,C 180,E1 -21878.278,E2 -21878.278} C_VEL
LIN {X 0,Y 196.094,Z 511.946,A -85,B 0,C 180,E1 -21881.363,E2 -21881.363} C_VEL
LIN {X 0,Y 197.761,Z 508.095,A -85,B 0,C 180,E1 -21884.399,E2 -21884.399} C_VEL
LIN {X 0,Y 199.921,Z 503.082,A -85,B 0,C 180,E1 -21887.38,E2 -21887.38} C_VEL
LIN {X 0,Y 202.552,Z 495.632,A -85,B 0,C 180,E1 -21890.827,E2 -21890.827} C_VEL
LIN {X 0,Y 205.201,Z 487.534,A -85,B 0,C 180,E1 -21893.724,E2 -21893.724} C_VEL
LIN {X 0,Y 207.298,Z 480.972,A -85,B 0,C 180,E1 -21895.605,E2 -21895.605} C_VEL
LIN {X 0,Y 209.381,Z 473.243,A -85,B 0,C 180,E1 -21897.48,E2 -21897.48} C_VEL
LIN {X 0,Y 211.951,Z 462.647,A -85,B 0,C 180,E1 -21899.547,E2 -21899.547} C_VEL
LIN {X 0,Y 214.215,Z 451.651,A -85,B 0,C 180,E1 -21901.208,E2 -21901.208} C_VEL
LIN {X 0,Y 215.461,Z 443.975,A -85,B 0,C 180,E1 -21902.16,E2 -21902.16} C_VEL
LIN {X 0,Y 212.702,Z 432.576,A -85,B 0,C 180,E1 -21904.082,E2 -21904.082} C_VEL
LIN {X 0,Y 208.642,Z 420.457,A -85,B 0,C 180,E1 -21905.953,E2 -21905.953} C_VEL
LIN {X 0,Y 204.594,Z 410.626,A -85,B 0,C 180,E1 -21907.355,E2 -21907.355} C_VEL
LIN {X 0,Y 204.952,Z 404.664,A -85,B 0,C 180,E1 -21910.649,E2 -21910.649} C_VEL
LIN {X 0,Y 204.404,Z 399.812,A -85,B 0,C 180,E1 -21913.776,E2 -21913.776} C_VEL
LIN {X 0,Y 203.665,Z 394.134,A -85,B 0,C 180,E1 -21917.708,E2 -21917.708} C_VEL
LIN {X 0,Y 202.599,Z 388.017,A -85,B 0,C 180,E1 -21922.192,E2 -21922.192} C_VEL
LIN {X 0,Y 201.621,Z 383.205,A -85,B 0,C 180,E1 -21926.101,E2 -21926.101} C_VEL
LIN {X 0,Y 200.363,Z 378.034,A -85,B 0,C 180,E1 -21930.588,E2 -21930.588} C_VEL
LIN {X 0,Y 199.287,Z 373.813,A -85,B 0,C 180,E1 -21934.963,E2 -21934.963} C_VEL
LIN {X 0,Y 197.793,Z 369.712,A -85,B 0,C 180,E1 -21939.186,E2 -21939.186} C_VEL
LIN {X 0,Y 196.697,Z 366.322,A -85,B 0,C 180,E1 -21943.39,E2 -21943.39} C_VEL
LIN {X 0,Y 196.139,Z 364.575,A -85,B 0,C 180,E1 -21945.473,E2 -21945.473} C_VEL
LIN {X 0,Y 195.107,Z 361.089,A -85,B 0,C 180,E1 -21951.715,E2 -21951.715} C_VEL
LIN {X 0,Y 193.607,Z 357.704,A -85,B 0,C 180,E1 -21959.999,E2 -21959.999} C_VEL
LIN {X 0,Y 193.39,Z 357.404,A -85,B 0,C 180,E1 -21962.082,E2 -21962.082} C_VEL
LIN {X 0,Y 193.147,Z 357.609,A -85,B 0,C 180,E1 -21964.695,E2 -21964.695} C_VEL
LIN {X 0,Y 194.32,Z 362.198,A -85,B 0,C 180,E1 -21969.366,E2 -21969.366} C_VEL
LIN {X 0,Y 195.575,Z 367.938,A -85,B 0,C 180,E1 -21974.568,E2 -21974.568} C_VEL
LIN {X 0,Y 197.106,Z 374.247,A -85,B 0,C 180,E1 -21979.799,E2 -21979.799} C_VEL
LIN {X 0,Y 198.494,Z 379.81,A -85,B 0,C 180,E1 -21984.027,E2 -21984.027} C_VEL
LIN {X 0,Y 200.465,Z 387.487,A -85,B 0,C 180,E1 -21989.394,E2 -21989.394} C_VEL
LIN {X 0,Y 202.26,Z 394.291,A -85,B 0,C 180,E1 -21993.776,E2 -21993.776} C_VEL
LIN {X 0,Y 204.246,Z 401.802,A -85,B 0,C 180,E1 -21998.269,E2 -21998.269} C_VEL
LIN {X 0,Y 205.638,Z 406.865,A -85,B 0,C 180,E1 -22001.131,E2 -22001.131} C_VEL
LIN {X 0,Y 213.796,Z 427.895,A -85,B 0,C 180,E1 -22003.654,E2 -22003.654} C_VEL
LIN {X 0,Y 214.658,Z 444.622,A -85,B 0,C 180,E1 -22005.297,E2 -22005.297} C_VEL
LIN {X 0,Y 215.354,Z 460.415,A -85,B 0,C 180,E1 -22007.191,E2 -22007.191} C_VEL
LIN {X 0,Y 215.839,Z 475.788,A -85,B 0,C 180,E1 -22009.373,E2 -22009.373} C_VEL
LIN {X 0,Y 215.419,Z 479.337,A -85,B 0,C 180,E1 -22009.891,E2 -22009.891} C_VEL
LIN {X 0,Y 211.605,Z 493.552,A -85,B 0,C 180,E1 -22012.096,E2 -22012.096} C_VEL
LIN {X 0,Y 208.185,Z 506.055,A -85,B 0,C 180,E1 -22014.471,E2 -22014.471} C_VEL
LIN {X 0,Y 205.233,Z 515.676,A -85,B 0,C 180,E1 -22016.613,E2 -22016.613} C_VEL
LIN {X 0,Y 203.397,Z 519.981,A -85,B 0,C 180,E1 -22017.665,E2 -22017.665} C_VEL
LIN {X 0,Y 198.601,Z 526.351,A -85,B 0,C 180,E1 -22019.419,E2 -22019.419} C_VEL
LIN {X 0,Y 194.677,Z 531.053,A -85,B 0,C 180,E1 -22020.891,E2 -22020.891} C_VEL
LIN {X 0,Y 192.507,Z 534.682,A -85,B 0,C 180,E1 -22022.06,E2 -22022.06} C_VEL
LIN {X 0,Y 192.06,Z 536.022,A -85,B 0,C 180,E1 -22022.45,E2 -22022.45} C_VEL
LIN {X 0,Y 189.808,Z 545.432,A -85,B 0,C 180,E1 -22025.389,E2 -22025.389} C_VEL
LIN {X 0,Y 187.973,Z 553.584,A -85,B 0,C 180,E1 -22028.578,E2 -22028.578} C_VEL
LIN {X 0,Y 186.81,Z 559.319,A -85,B 0,C 180,E1 -22031.356,E2 -22031.356} C_VEL
LIN {X 0,Y 185.82,Z 564.848,A -85,B 0,C 180,E1 -22034.654,E2 -22034.654} C_VEL
LIN {X 0,Y 185.328,Z 569.171,A -85,B 0,C 180,E1 -22037.967,E2 -22037.967} C_VEL
LIN {X 0,Y 185.29,Z 572.411,A -85,B 0,C 180,E1 -22041.279,E2 -22041.279} C_VEL
LIN {X 0,Y 185.346,Z 573.977,A -85,B 0,C 180,E1 -22043.474,E2 -22043.474} C_VEL
LIN {X 0,Y 185.5,Z 575.1,A -85,B 0,C 180,E1 -22045.66,E2 -22045.66} C_VEL
LIN {X 0,Y 185.75,Z 575.808,A -85,B 0,C 180,E1 -22047.837,E2 -22047.837} C_VEL
LIN {X 0,Y 185.991,Z 576.079,A -85,B 0,C 180,E1 -22050.005,E2 -22050.005} C_VEL
LIN {X 0,Y 185.792,Z 575.816,A -85,B 0,C 180,E1 -22052.173,E2 -22052.173} C_VEL
LIN {X 0,Y 185.528,Z 575.91,A -85,B 0,C 180,E1 -22054.35,E2 -22054.35} C_VEL
LIN {X 0,Y 184.823,Z 575.589,A -85,B 0,C 180,E1 -22058.754,E2 -22058.754} C_VEL
LIN {X 0,Y 184.758,Z 574.267,A -85,B 0,C 180,E1 -22063.198,E2 -22063.198} C_VEL
LIN {X 0,Y 186.077,Z 571.117,A -85,B 0,C 180,E1 -22069.228,E2 -22069.228} C_VEL
LIN {X 0,Y 188.587,Z 567.371,A -85,B 0,C 180,E1 -22074.206,E2 -22074.206} C_VEL
LIN {X 0,Y 194.151,Z 560.952,A -85,B 0,C 180,E1 -22080.455,E2 -22080.455} C_VEL
LIN {X 0,Y 200.724,Z 554.374,A -85,B 0,C 180,E1 -22085.295,E2 -22085.295} C_VEL
LIN {X 0,Y 210.711,Z 545.126,A -85,B 0,C 180,E1 -22090.577,E2 -22090.577} C_VEL
LIN {X 0,Y 220.737,Z 536.253,A -85,B 0,C 180,E1 -22094.468,E2 -22094.468} C_VEL
LIN {X 0,Y 229.688,Z 528.443,A -85,B 0,C 180,E1 -22097.257,E2 -22097.257} C_VEL
LIN {X 0,Y 244.835,Z 515.224,A -85,B 0,C 180,E1 -22100.813,E2 -22100.813} C_VEL
LIN {X 0,Y 248.564,Z 511.868,A -85,B 0,C 180,E1 -22101.546,E2 -22101.546} C_VEL
LIN {X 0,Y 248.447,Z 511.657,A -85,B 0,C 180,E1 -22102.03,E2 -22102.03} C_VEL
LIN {X 0,Y 237.544,Z 518.158,A -85,B 0,C 180,E1 -22104.766,E2 -22104.766} C_VEL
LIN {X 0,Y 226.6,Z 523.889,A -85,B 0,C 180,E1 -22108.181,E2 -22108.181} C_VEL
LIN {X 0,Y 218.658,Z 527.368,A -85,B 0,C 180,E1 -22111.177,E2 -22111.177} C_VEL
LIN {X 0,Y 211.528,Z 529.865,A -85,B 0,C 180,E1 -22114.411,E2 -22114.411} C_VEL
LIN {X 0,Y 205.233,Z 531.343,A -85,B 0,C 180,E1 -22117.872,E2 -22117.872} C_VEL
LIN {X 0,Y 199.813,Z 531.737,A -85,B 0,C 180,E1 -22121.546,E2 -22121.546} C_VEL
LIN {X 0,Y 195.374,Z 530.963,A -85,B 0,C 180,E1 -22125.417,E2 -22125.417} C_VEL
LIN {X 0,Y 191.97,Z 528.931,A -85,B 0,C 180,E1 -22129.453,E2 -22129.453} C_VEL
LIN {X 0,Y 189.38,Z 525.599,A -85,B 0,C 180,E1 -22133.609,E2 -22133.609} C_VEL
LIN {X 0,Y 187.537,Z 520.874,A -85,B 0,C 180,E1 -22137.853,E2 -22137.853} C_VEL
LIN {X 0,Y 186.691,Z 514.636,A -85,B 0,C 180,E1 -22142.158,E2 -22142.158} C_VEL
LIN {X 0,Y 186.515,Z 506.651,A -85,B 0,C 180,E1 -22146.492,E2 -22146.492} C_VEL
LIN {X 0,Y 187.07,Z 498.12,A -85,B 0,C 180,E1 -22150.28,E2 -22150.28} C_VEL
LIN {X 0,Y 188.164,Z 488.623,A -85,B 0,C 180,E1 -22153.79,E2 -22153.79} C_VEL
LIN {X 0,Y 189.627,Z 477.501,A -85,B 0,C 180,E1 -22157.248,E2 -22157.248} C_VEL
LIN {X 0,Y 191.471,Z 465.213,A -85,B 0,C 180,E1 -22160.409,E2 -22160.409} C_VEL
LIN {X 0,Y 193.576,Z 451.976,A -85,B 0,C 180,E1 -22163.256,E2 -22163.256} C_VEL
LIN {X 0,Y 195.763,Z 437.56,A -85,B 0,C 180,E1 -22165.824,E2 -22165.824} C_VEL
LIN {X 0,Y 197.138,Z 425.832,A -85,B 0,C 180,E1 -22167.611,E2 -22167.611} C_VEL
LIN {X 0,Y 194.611,Z 411.008,A -85,B 0,C 180,E1 -22169.913,E2 -22169.913} C_VEL
LIN {X 0,Y 191.464,Z 395.662,A -85,B 0,C 180,E1 -22172.025,E2 -22172.025} C_VEL
LIN {X 0,Y 190.15,Z 389.347,A -85,B 0,C 180,E1 -22172.847,E2 -22172.847} C_VEL
LIN {X 0,Y 191.183,Z 389.399,A -85,B 0,C 180,E1 -22173.465,E2 -22173.465} C_VEL
LIN {X 0,Y 193.216,Z 390.777,A -85,B 0,C 180,E1 -22175.591,E2 -22175.591} C_VEL
LIN {X 0,Y 195.034,Z 392.524,A -85,B 0,C 180,E1 -22177.778,E2 -22177.778} C_VEL
LIN {X 0,Y 196.459,Z 394.935,A -85,B 0,C 180,E1 -22180.086,E2 -22180.086} C_VEL
LIN {X 0,Y 197.423,Z 397.939,A -85,B 0,C 180,E1 -22182.562,E2 -22182.562} C_VEL
LIN {X 0,Y 198.171,Z 403,A -85,B 0,C 180,E1 -22186.138,E2 -22186.138} C_VEL
LIN {X 0,Y 198.657,Z 407.816,A -85,B 0,C 180,E1 -22189.238,E2 -22189.238} C_VEL
LIN {X 0,Y 198.43,Z 411.935,A -85,B 0,C 180,E1 -22191.456,E2 -22191.456} C_VEL
LIN {X 0,Y 203.148,Z 423.601,A -85,B 0,C 180,E1 -22193.237,E2 -22193.237} C_VEL
LIN {X 0,Y 206.827,Z 434.995,A -85,B 0,C 180,E1 -22195.112,E2 -22195.112} C_VEL
LIN {X 0,Y 209.221,Z 445.067,A -85,B 0,C 180,E1 -22196.912,E2 -22196.912} C_VEL
LIN {X 0,Y 208.481,Z 450.91,A -85,B 0,C 180,E1 -22197.682,E2 -22197.682} C_VEL
LIN {X 0,Y 205.974,Z 462.923,A -85,B 0,C 180,E1 -22199.495,E2 -22199.495} C_VEL
LIN {X 0,Y 203.253,Z 473.713,A -85,B 0,C 180,E1 -22201.607,E2 -22201.607} C_VEL
LIN {X 0,Y 201.154,Z 481.514,A -85,B 0,C 180,E1 -22203.542,E2 -22203.542} C_VEL
LIN {X 0,Y 198.436,Z 489.651,A -85,B 0,C 180,E1 -22205.96,E2 -22205.96} C_VEL
LIN {X 0,Y 195.609,Z 497.555,A -85,B 0,C 180,E1 -22208.939,E2 -22208.939} C_VEL
LIN {X 0,Y 193.271,Z 503.88,A -85,B 0,C 180,E1 -22211.991,E2 -22211.991} C_VEL
LIN {X 0,Y 190.998,Z 508.95,A -85,B 0,C 180,E1 -22215.069,E2 -22215.069} C_VEL
LIN {X 0,Y 189.242,Z 512.857,A -85,B 0,C 180,E1 -22218.209,E2 -22218.209} C_VEL
LIN {X 0,Y 188.197,Z 515.688,A -85,B 0,C 180,E1 -22221.404,E2 -22221.404} C_VEL
LIN {X 0,Y 187.669,Z 517.061,A -85,B 0,C 180,E1 -22223.544,E2 -22223.544} C_VEL
LIN {X 0,Y 186.997,Z 518.626,A -85,B 0,C 180,E1 -22227.841,E2 -22227.841} C_VEL
LIN {X 0,Y 186.913,Z 518.852,A -85,B 0,C 180,E1 -22229.995,E2 -22229.995} C_VEL
LIN {X 0,Y 187.278,Z 518.078,A -85,B 0,C 180,E1 -22234.299,E2 -22234.299} C_VEL
LIN {X 0,Y 187.677,Z 517.134,A -85,B 0,C 180,E1 -22236.445,E2 -22236.445} C_VEL
LIN {X 0,Y 188.188,Z 515.807,A -85,B 0,C 180,E1 -22238.586,E2 -22238.586} C_VEL
LIN {X 0,Y 189.216,Z 513.022,A -85,B 0,C 180,E1 -22241.782,E2 -22241.782} C_VEL
LIN {X 0,Y 190.972,Z 509.169,A -85,B 0,C 180,E1 -22244.923,E2 -22244.923} C_VEL
LIN {X 0,Y 193.239,Z 504.155,A -85,B 0,C 180,E1 -22248.002,E2 -22248.002} C_VEL
LIN {X 0,Y 196.015,Z 496.702,A -85,B 0,C 180,E1 -22251.556,E2 -22251.556} C_VEL
LIN {X 0,Y 198.796,Z 488.602,A -85,B 0,C 180,E1 -22254.538,E2 -22254.538} C_VEL
LIN {X 0,Y 200.989,Z 482.039,A -85,B 0,C 180,E1 -22256.47,E2 -22256.47} C_VEL
LIN {X 0,Y 203.179,Z 474.307,A -85,B 0,C 180,E1 -22258.393,E2 -22258.393} C_VEL
LIN {X 0,Y 205.872,Z 463.705,A -85,B 0,C 180,E1 -22260.511,E2 -22260.511} C_VEL
LIN {X 0,Y 208.454,Z 451.6,A -85,B 0,C 180,E1 -22262.357,E2 -22262.357} C_VEL
LIN {X 0,Y 209.416,Z 446.117,A -85,B 0,C 180,E1 -22263.042,E2 -22263.042} C_VEL
LIN {X 0,Y 207.079,Z 435.707,A -85,B 0,C 180,E1 -22264.911,E2 -22264.911} C_VEL
LIN {X 0,Y 203.371,Z 423.948,A -85,B 0,C 180,E1 -22266.847,E2 -22266.847} C_VEL
LIN {X 0,Y 198.422,Z 411.68,A -85,B 0,C 180,E1 -22268.749,E2 -22268.749} C_VEL
LIN {X 0,Y 198.678,Z 408.142,A -85,B 0,C 180,E1 -22270.756,E2 -22270.756} C_VEL
LIN {X 0,Y 198.243,Z 403.385,A -85,B 0,C 180,E1 -22273.868,E2 -22273.868} C_VEL
LIN {X 0,Y 197.373,Z 396.901,A -85,B 0,C 180,E1 -22278.388,E2 -22278.388} C_VEL
LIN {X 0,Y 196.556,Z 391.53,A -85,B 0,C 180,E1 -22282.565,E2 -22282.565} C_VEL
LIN {X 0,Y 195.59,Z 386.634,A -85,B 0,C 180,E1 -22286.619,E2 -22286.619} C_VEL
LIN {X 0,Y 194.407,Z 381.564,A -85,B 0,C 180,E1 -22291.194,E2 -22291.194} C_VEL
LIN {X 0,Y 193.492,Z 377.836,A -85,B 0,C 180,E1 -22295.222,E2 -22295.222} C_VEL
LIN {X 0,Y 192.576,Z 374.905,A -85,B 0,C 180,E1 -22298.595,E2 -22298.595} C_VEL
LIN {X 0,Y 191.319,Z 371.243,A -85,B 0,C 180,E1 -22302.909,E2 -22302.909} C_VEL
LIN {X 0,Y 190.939,Z 369.707,A -85,B 0,C 180,E1 -22305.068,E2 -22305.068} C_VEL
LIN {X 0,Y 189.844,Z 366.031,A -85,B 0,C 180,E1 -22311.484,E2 -22311.484} C_VEL
LIN {X 0,Y 189.082,Z 364.677,A -85,B 0,C 180,E1 -22315.736,E2 -22315.736} C_VEL
LIN {X 0,Y 188.794,Z 362.957,A -85,B 0,C 180,E1 -22319.999,E2 -22319.999} C_VEL
LIN {X 0,Y 188.587,Z 362.649,A -85,B 0,C 180,E1 -22322.135,E2 -22322.135} C_VEL
LIN {X 0,Y 188.342,Z 362.67,A -85,B 0,C 180,E1 -22324.279,E2 -22324.279} C_VEL
LIN {X 0,Y 187.708,Z 364.995,A -85,B 0,C 180,E1 -22329.699,E2 -22329.699} C_VEL
LIN {X 0,Y 189.004,Z 370.848,A -85,B 0,C 180,E1 -22335.086,E2 -22335.086} C_VEL
LIN {X 0,Y 190.58,Z 377.314,A -85,B 0,C 180,E1 -22340.507,E2 -22340.507} C_VEL
LIN {X 0,Y 191.976,Z 383.038,A -85,B 0,C 180,E1 -22344.897,E2 -22344.897} C_VEL
LIN {X 0,Y 193.646,Z 389.411,A -85,B 0,C 180,E1 -22349.434,E2 -22349.434} C_VEL
LIN {X 0,Y 195.896,Z 397.954,A -85,B 0,C 180,E1 -22355.03,E2 -22355.03} C_VEL
LIN {X 0,Y 197.6,Z 404.356,A -85,B 0,C 180,E1 -22358.845,E2 -22358.845} C_VEL
LIN {X 0,Y 198.776,Z 408.426,A -85,B 0,C 180,E1 -22360.35,E2 -22360.35} C_VEL
LIN {X 0,Y 207.092,Z 429.392,A -85,B 0,C 180,E1 -22363.011,E2 -22363.011} C_VEL
LIN {X 0,Y 207.865,Z 442.511,A -85,B 0,C 180,E1 -22364.365,E2 -22364.365} C_VEL
LIN {X 0,Y 208.473,Z 459.501,A -85,B 0,C 180,E1 -22366.451,E2 -22366.451} C_VEL
LIN {X 0,Y 208.951,Z 474.866,A -85,B 0,C 180,E1 -22368.701,E2 -22368.701} C_VEL
LIN {X 0,Y 208.714,Z 478.621,A -85,B 0,C 180,E1 -22369.284,E2 -22369.284} C_VEL
LIN {X 0,Y 204.848,Z 492.772,A -85,B 0,C 180,E1 -22371.557,E2 -22371.557} C_VEL
LIN {X 0,Y 201.089,Z 506.014,A -85,B 0,C 180,E1 -22374.175,E2 -22374.175} C_VEL
LIN {X 0,Y 197.322,Z 518.222,A -85,B 0,C 180,E1 -22377.108,E2 -22377.108} C_VEL
LIN {X 0,Y 193.83,Z 529.761,A -85,B 0,C 180,E1 -22380.481,E2 -22380.481} C_VEL
LIN {X 0,Y 192.06,Z 536.022,A -85,B 0,C 180,E1 -22382.45,E2 -22382.45} C_VEL
LIN {X 0,Y 190.387,Z 540.22,A -85,B 0,C 180,E1 -22383.611,E2 -22383.611} C_VEL
LIN {X 0,Y 186.101,Z 546.58,A -85,B 0,C 180,E1 -22385.534,E2 -22385.534} C_VEL
LIN {X 0,Y 181.954,Z 552.278,A -85,B 0,C 180,E1 -22387.69,E2 -22387.69} C_VEL
LIN {X 0,Y 180.532,Z 555.485,A -85,B 0,C 180,E1 -22389.183,E2 -22389.183} C_VEL
LIN {X 0,Y 179.196,Z 562.031,A -85,B 0,C 180,E1 -22392.9,E2 -22392.9} C_VEL
LIN {X 0,Y 178.416,Z 566.731,A -85,B 0,C 180,E1 -22396.335,E2 -22396.335} C_VEL
LIN {X 0,Y 178.218,Z 570.821,A -85,B 0,C 180,E1 -22400.352,E2 -22400.352} C_VEL
LIN {X 0,Y 178.293,Z 572.888,A -85,B 0,C 180,E1 -22403.214,E2 -22403.214} C_VEL
LIN {X 0,Y 178.437,Z 574.013,A -85,B 0,C 180,E1 -22405.488,E2 -22405.488} C_VEL
LIN {X 0,Y 178.699,Z 574.725,A -85,B 0,C 180,E1 -22407.752,E2 -22407.752} C_VEL
LIN {X 0,Y 178.986,Z 575.004,A -85,B 0,C 180,E1 -22410.005,E2 -22410.005} C_VEL
LIN {X 0,Y 178.557,Z 574.341,A -85,B 0,C 180,E1 -22414.52,E2 -22414.52} C_VEL
LIN {X 0,Y 177.813,Z 574.131,A -85,B 0,C 180,E1 -22419.102,E2 -22419.102} C_VEL
LIN {X 0,Y 177.779,Z 572.982,A -85,B 0,C 180,E1 -22423.726,E2 -22423.726} C_VEL
LIN {X 0,Y 179.153,Z 570.251,A -85,B 0,C 180,E1 -22429.698,E2 -22429.698} C_VEL
LIN {X 0,Y 181.989,Z 566.491,A -85,B 0,C 180,E1 -22435.143,E2 -22435.143} C_VEL
LIN {X 0,Y 187.945,Z 560.434,A -85,B 0,C 180,E1 -22441.574,E2 -22441.574} C_VEL
LIN {X 0,Y 196.46,Z 552.883,A -85,B 0,C 180,E1 -22447.461,E2 -22447.461} C_VEL
LIN {X 0,Y 207.315,Z 543.919,A -85,B 0,C 180,E1 -22452.693,E2 -22452.693} C_VEL
LIN {X 0,Y 220.224,Z 533.559,A -85,B 0,C 180,E1 -22457.228,E2 -22457.228} C_VEL
LIN {X 0,Y 231.361,Z 524.815,A -85,B 0,C 180,E1 -22460.091,E2 -22460.091} C_VEL
LIN {X 0,Y 238.388,Z 519.18,A -85,B 0,C 180,E1 -22461.639,E2 -22461.639} C_VEL
LIN {X 0,Y 239.773,Z 517.981,A -85,B 0,C 180,E1 -22462.01,E2 -22462.01} C_VEL
LIN {X 0,Y 230.057,Z 522.924,A -85,B 0,C 180,E1 -22464.52,E2 -22464.52} C_VEL
LIN {X 0,Y 221.088,Z 526.96,A -85,B 0,C 180,E1 -22467.29,E2 -22467.29} C_VEL
LIN {X 0,Y 212.89,Z 530.038,A -85,B 0,C 180,E1 -22470.319,E2 -22470.319} C_VEL
LIN {X 0,Y 205.486,Z 532.175,A -85,B 0,C 180,E1 -22473.602,E2 -22473.602} C_VEL
LIN {X 0,Y 198.942,Z 533.298,A -85,B 0,C 180,E1 -22477.134,E2 -22477.134} C_VEL
LIN {X 0,Y 193.28,Z 533.349,A -85,B 0,C 180,E1 -22480.899,E2 -22480.899} C_VEL
LIN {X 0,Y 188.649,Z 532.25,A -85,B 0,C 180,E1 -22484.885,E2 -22484.885} C_VEL
LIN {X 0,Y 185.075,Z 529.927,A -85,B 0,C 180,E1 -22489.056,E2 -22489.056} C_VEL
LIN {X 0,Y 182.371,Z 526.311,A -85,B 0,C 180,E1 -22493.362,E2 -22493.362} C_VEL
LIN {X 0,Y 180.462,Z 521.309,A -85,B 0,C 180,E1 -22497.769,E2 -22497.769} C_VEL
LIN {X 0,Y 179.584,Z 514.739,A -85,B 0,C 180,E1 -22502.244,E2 -22502.244} C_VEL
LIN {X 0,Y 179.437,Z 507.629,A -85,B 0,C 180,E1 -22506.184,E2 -22506.184} C_VEL
LIN {X 0,Y 180.008,Z 498.296,A -85,B 0,C 180,E1 -22510.444,E2 -22510.444} C_VEL
LIN {X 0,Y 180.906,Z 490.371,A -85,B 0,C 180,E1 -22513.48,E2 -22513.48} C_VEL
LIN {X 0,Y 182.229,Z 480.199,A -85,B 0,C 180,E1 -22516.814,E2 -22516.814} C_VEL
LIN {X 0,Y 184.233,Z 467.232,A -85,B 0,C 180,E1 -22520.372,E2 -22520.372} C_VEL
LIN {X 0,Y 186.33,Z 454.219,A -85,B 0,C 180,E1 -22523.332,E2 -22523.332} C_VEL
LIN {X 0,Y 188.583,Z 440.212,A -85,B 0,C 180,E1 -22525.97,E2 -22525.97} C_VEL
LIN {X 0,Y 190.206,Z 428.513,A -85,B 0,C 180,E1 -22527.841,E2 -22527.841} C_VEL
LIN {X 0,Y 189.795,Z 423.68,A -85,B 0,C 180,E1 -22528.631,E2 -22528.631} C_VEL
LIN {X 0,Y 187.27,Z 409.163,A -85,B 0,C 180,E1 -22530.926,E2 -22530.926} C_VEL
LIN {X 0,Y 184.163,Z 393.932,A -85,B 0,C 180,E1 -22533.084,E2 -22533.084} C_VEL
LIN {X 0,Y 186.26,Z 394.136,A -85,B 0,C 180,E1 -22534.472,E2 -22534.472} C_VEL
LIN {X 0,Y 188.225,Z 395.64,A -85,B 0,C 180,E1 -22536.686,E2 -22536.686} C_VEL
LIN {X 0,Y 189.899,Z 397.634,A -85,B 0,C 180,E1 -22538.989,E2 -22538.989} C_VEL
LIN {X 0,Y 191.089,Z 400.365,A -85,B 0,C 180,E1 -22541.455,E2 -22541.455} C_VEL
LIN {X 0,Y 191.871,Z 405.404,A -85,B 0,C 180,E1 -22545.199,E2 -22545.199} C_VEL
LIN {X 0,Y 192.379,Z 410.888,A -85,B 0,C 180,E1 -22548.879,E2 -22548.879} C_VEL
LIN {X 0,Y 192.266,Z 412.877,A -85,B 0,C 180,E1 -22549.969,E2 -22549.969} C_VEL
LIN {X 0,Y 197.307,Z 425.302,A -85,B 0,C 180,E1 -22552.008,E2 -22552.008} C_VEL
LIN {X 0,Y 200.875,Z 436.758,A -85,B 0,C 180,E1 -22553.998,E2 -22553.998} C_VEL
LIN {X 0,Y 203.132,Z 446.512,A -85,B 0,C 180,E1 -22555.839,E2 -22555.839} C_VEL
LIN {X 0,Y 203.298,Z 447.694,A -85,B 0,C 180,E1 -22556.067,E2 -22556.067} C_VEL
LIN {X 0,Y 201.001,Z 459.555,A -85,B 0,C 180,E1 -22557.73,E2 -22557.73} C_VEL
LIN {X 0,Y 198.389,Z 470.302,A -85,B 0,C 180,E1 -22559.676,E2 -22559.676} C_VEL
LIN {X 0,Y 195.863,Z 478.875,A -85,B 0,C 180,E1 -22561.607,E2 -22561.607} C_VEL
LIN {X 0,Y 193.696,Z 486.037,A -85,B 0,C 180,E1 -22563.605,E2 -22563.605} C_VEL
LIN {X 0,Y 190.485,Z 494.898,A -85,B 0,C 180,E1 -22566.628,E2 -22566.628} C_VEL
LIN {X 0,Y 188.106,Z 501.27,A -85,B 0,C 180,E1 -22569.407,E2 -22569.407} C_VEL
LIN {X 0,Y 185.809,Z 506.763,A -85,B 0,C 180,E1 -22572.382,E2 -22572.382} C_VEL
LIN {X 0,Y 183.581,Z 511.427,A -85,B 0,C 180,E1 -22575.586,E2 -22575.586} C_VEL
LIN {X 0,Y 181.985,Z 514.963,A -85,B 0,C 180,E1 -22578.861,E2 -22578.861} C_VEL
LIN {X 0,Y 181.259,Z 516.766,A -85,B 0,C 180,E1 -22581.073,E2 -22581.073} C_VEL
LIN {X 0,Y 180.702,Z 518.137,A -85,B 0,C 180,E1 -22583.294,E2 -22583.294} C_VEL
LIN {X 0,Y 179.984,Z 519.703,A -85,B 0,C 180,E1 -22587.757,E2 -22587.757} C_VEL
LIN {X 0,Y 179.911,Z 519.926,A -85,B 0,C 180,E1 -22589.995,E2 -22589.995} C_VEL
LIN {X 0,Y 180.288,Z 519.154,A -85,B 0,C 180,E1 -22594.466,E2 -22594.466} C_VEL
LIN {X 0,Y 180.731,Z 518.206,A -85,B 0,C 180,E1 -22596.694,E2 -22596.694} C_VEL
LIN {X 0,Y 181.25,Z 516.883,A -85,B 0,C 180,E1 -22598.917,E2 -22598.917} C_VEL
LIN {X 0,Y 182.35,Z 514.097,A -85,B 0,C 180,E1 -22602.232,E2 -22602.232} C_VEL
LIN {X 0,Y 184.2,Z 510.243,A -85,B 0,C 180,E1 -22605.485,E2 -22605.485} C_VEL
LIN {X 0,Y 186.58,Z 505.227,A -85,B 0,C 180,E1 -22608.668,E2 -22608.668} C_VEL
LIN {X 0,Y 189.529,Z 497.77,A -85,B 0,C 180,E1 -22612.333,E2 -22612.333} C_VEL
LIN {X 0,Y 192.433,Z 489.671,A -85,B 0,C 180,E1 -22615.406,E2 -22615.406} C_VEL
LIN {X 0,Y 194.729,Z 483.106,A -85,B 0,C 180,E1 -22617.391,E2 -22617.391} C_VEL
LIN {X 0,Y 197.031,Z 475.371,A -85,B 0,C 180,E1 -22619.364,E2 -22619.364} C_VEL
LIN {X 0,Y 199.855,Z 464.762,A -85,B 0,C 180,E1 -22621.533,E2 -22621.533} C_VEL
LIN {X 0,Y 202.519,Z 452.922,A -85,B 0,C 180,E1 -22623.379,E2 -22623.379} C_VEL
LIN {X 0,Y 203.274,Z 448.765,A -85,B 0,C 180,E1 -22623.923,E2 -22623.923} C_VEL
LIN {X 0,Y 202.955,Z 445.338,A -85,B 0,C 180,E1 -22624.533,E2 -22624.533} C_VEL
LIN {X 0,Y 200.15,Z 433.976,A -85,B 0,C 180,E1 -22626.643,E2 -22626.643} C_VEL
LIN {X 0,Y 196.468,Z 422.822,A -85,B 0,C 180,E1 -22628.556,E2 -22628.556} C_VEL
LIN {X 0,Y 192.312,Z 412.747,A -85,B 0,C 180,E1 -22630.246,E2 -22630.246} C_VEL
LIN {X 0,Y 192.35,Z 409.418,A -85,B 0,C 180,E1 -22632.313,E2 -22632.313} C_VEL
LIN {X 0,Y 191.53,Z 402.382,A -85,B 0,C 180,E1 -22637.204,E2 -22637.204} C_VEL
LIN {X 0,Y 190.795,Z 397.093,A -85,B 0,C 180,E1 -22641.229,E2 -22641.229} C_VEL
LIN {X 0,Y 189.965,Z 392.152,A -85,B 0,C 180,E1 -22645.338,E2 -22645.338} C_VEL
LIN {X 0,Y 189.028,Z 387.285,A -85,B 0,C 180,E1 -22649.803,E2 -22649.803} C_VEL
LIN {X 0,Y 188.101,Z 383.389,A -85,B 0,C 180,E1 -22653.715,E2 -22653.715} C_VEL
LIN {X 0,Y 187.224,Z 379.99,A -85,B 0,C 180,E1 -22657.951,E2 -22657.951} C_VEL
LIN {X 0,Y 186.072,Z 376.348,A -85,B 0,C 180,E1 -22662.412,E2 -22662.412} C_VEL
LIN {X 0,Y 185.422,Z 373.571,A -85,B 0,C 180,E1 -22666.854,E2 -22666.854} C_VEL
LIN {X 0,Y 184.615,Z 370.81,A -85,B 0,C 180,E1 -22671.754,E2 -22671.754} C_VEL
LIN {X 0,Y 184.048,Z 369,A -85,B 0,C 180,E1 -22677.811,E2 -22677.811} C_VEL
LIN {X 0,Y 183.999,Z 368.191,A -85,B 0,C 180,E1 -22679.999,E2 -22679.999} C_VEL
LIN {X 0,Y 183.843,Z 367.946,A -85,B 0,C 180,E1 -22682.19,E2 -22682.19} C_VEL
LIN {X 0,Y 183.705,Z 368.202,A -85,B 0,C 180,E1 -22684.387,E2 -22684.387} C_VEL
LIN {X 0,Y 183.13,Z 369.928,A -85,B 0,C 180,E1 -22688.829,E2 -22688.829} C_VEL
LIN {X 0,Y 182.946,Z 375.304,A -85,B 0,C 180,E1 -22696.204,E2 -22696.204} C_VEL
LIN {X 0,Y 183.69,Z 378.992,A -85,B 0,C 180,E1 -22700.141,E2 -22700.141} C_VEL
LIN {X 0,Y 185.1,Z 384.742,A -85,B 0,C 180,E1 -22704.686,E2 -22704.686} C_VEL
LIN {X 0,Y 186.758,Z 391.061,A -85,B 0,C 180,E1 -22709.288,E2 -22709.288} C_VEL
LIN {X 0,Y 189.694,Z 401.127,A -85,B 0,C 180,E1 -22714.609,E2 -22714.609} C_VEL
LIN {X 0,Y 192.554,Z 409.094,A -85,B 0,C 180,E1 -22718.35,E2 -22718.35} C_VEL
LIN {X 0,Y 193.715,Z 413.831,A -85,B 0,C 180,E1 -22720.084,E2 -22720.084} C_VEL
LIN {X 0,Y 200.743,Z 432.127,A -85,B 0,C 180,E1 -22722.519,E2 -22722.519} C_VEL
LIN {X 0,Y 201.368,Z 450.081,A -85,B 0,C 180,E1 -22724.564,E2 -22724.564} C_VEL
LIN {X 0,Y 201.873,Z 465.995,A -85,B 0,C 180,E1 -22726.767,E2 -22726.767} C_VEL
LIN {X 0,Y 202.01,Z 477.699,A -85,B 0,C 180,E1 -22728.63,E2 -22728.63} C_VEL
LIN {X 0,Y 198.273,Z 491.385,A -85,B 0,C 180,E1 -22730.9,E2 -22730.9} C_VEL
LIN {X 0,Y 194.289,Z 505.054,A -85,B 0,C 180,E1 -22733.685,E2 -22733.685} C_VEL
LIN {X 0,Y 190.146,Z 518.15,A -85,B 0,C 180,E1 -22736.97,E2 -22736.97} C_VEL
LIN {X 0,Y 188.239,Z 524.302,A -85,B 0,C 180,E1 -22738.714,E2 -22738.714} C_VEL
LIN {X 0,Y 185.883,Z 534.132,A -85,B 0,C 180,E1 -22741.187,E2 -22741.187} C_VEL
LIN {X 0,Y 183.587,Z 542.782,A -85,B 0,C 180,E1 -22743.888,E2 -22743.888} C_VEL
LIN {X 0,Y 181.449,Z 551.291,A -85,B 0,C 180,E1 -22747.218,E2 -22747.218} C_VEL
LIN {X 0,Y 180.532,Z 555.485,A -85,B 0,C 180,E1 -22749.183,E2 -22749.183} C_VEL
LIN {X 0,Y 179.173,Z 558.489,A -85,B 0,C 180,E1 -22750.752,E2 -22750.752} C_VEL
LIN {X 0,Y 175.425,Z 562.715,A -85,B 0,C 180,E1 -22753.394,E2 -22753.394} C_VEL
LIN {X 0,Y 172.539,Z 565.572,A -85,B 0,C 180,E1 -22755.656,E2 -22755.656} C_VEL
LIN {X 0,Y 171.301,Z 567.489,A -85,B 0,C 180,E1 -22757.48,E2 -22757.48} C_VEL
LIN {X 0,Y 171.183,Z 568.089,A -85,B 0,C 180,E1 -22758.106,E2 -22758.106} C_VEL
LIN {X 0,Y 171.168,Z 570.219,A -85,B 0,C 180,E1 -22760.553,E2 -22760.553} C_VEL
LIN {X 0,Y 171.242,Z 571.799,A -85,B 0,C 180,E1 -22762.934,E2 -22762.934} C_VEL
LIN {X 0,Y 171.374,Z 572.927,A -85,B 0,C 180,E1 -22765.301,E2 -22765.301} C_VEL
LIN {X 0,Y 171.645,Z 573.642,A -85,B 0,C 180,E1 -22767.659,E2 -22767.659} C_VEL
LIN {X 0,Y 171.976,Z 573.928,A -85,B 0,C 180,E1 -22770.006,E2 -22770.006} C_VEL
LIN {X 0,Y 171.753,Z 573.647,A -85,B 0,C 180,E1 -22772.351,E2 -22772.351} C_VEL
LIN {X 0,Y 171.542,Z 572.947,A -85,B 0,C 180,E1 -22774.706,E2 -22774.706} C_VEL
LIN {X 0,Y 170.82,Z 572.613,A -85,B 0,C 180,E1 -22779.478,E2 -22779.478} C_VEL
LIN {X 0,Y 170.827,Z 571.619,A -85,B 0,C 180,E1 -22784.297,E2 -22784.297} C_VEL
LIN {X 0,Y 172.249,Z 569.226,A -85,B 0,C 180,E1 -22790.213,E2 -22790.213} C_VEL
LIN {X 0,Y 175.445,Z 565.625,A -85,B 0,C 180,E1 -22796.15,E2 -22796.15} C_VEL
LIN {X 0,Y 181.813,Z 559.943,A -85,B 0,C 180,E1 -22802.769,E2 -22802.769} C_VEL
LIN {X 0,Y 190.798,Z 552.835,A -85,B 0,C 180,E1 -22808.775,E2 -22808.775} C_VEL
LIN {X 0,Y 202.136,Z 544.388,A -85,B 0,C 180,E1 -22814.062,E2 -22814.062} C_VEL
LIN {X 0,Y 215.522,Z 534.651,A -85,B 0,C 180,E1 -22818.597,E2 -22818.597} C_VEL
LIN {X 0,Y 227.921,Z 525.718,A -85,B 0,C 180,E1 -22821.64,E2 -22821.64} C_VEL
LIN {X 0,Y 229.74,Z 524.238,A -85,B 0,C 180,E1 -22822.279,E2 -22822.279} C_VEL
LIN {X 0,Y 220.16,Z 528.257,A -85,B 0,C 180,E1 -22824.929,E2 -22824.929} C_VEL
LIN {X 0,Y 211.277,Z 531.412,A -85,B 0,C 180,E1 -22827.845,E2 -22827.845} C_VEL
LIN {X 0,Y 203.172,Z 533.617,A -85,B 0,C 180,E1 -22831.036,E2 -22831.036} C_VEL
LIN {X 0,Y 195.932,Z 534.873,A -85,B 0,C 180,E1 -22834.506,E2 -22834.506} C_VEL
LIN {X 0,Y 189.567,Z 535.132,A -85,B 0,C 180,E1 -22838.24,E2 -22838.24} C_VEL
LIN {X 0,Y 184.195,Z 534.302,A -85,B 0,C 180,E1 -22842.228,E2 -22842.228} C_VEL
LIN {X 0,Y 179.917,Z 532.292,A -85,B 0,C 180,E1 -22846.446,E2 -22846.446} C_VEL
LIN {X 0,Y 176.576,Z 529.031,A -85,B 0,C 180,E1 -22850.84,E2 -22850.84} C_VEL
LIN {X 0,Y 174.709,Z 525.73,A -85,B 0,C 180,E1 -22854.229,E2 -22854.229} C_VEL
LIN {X 0,Y 173.078,Z 520.081,A -85,B 0,C 180,E1 -22858.838,E2 -22858.838} C_VEL
LIN {X 0,Y 172.385,Z 512.808,A -85,B 0,C 180,E1 -22863.507,E2 -22863.507} C_VEL
LIN {X 0,Y 172.417,Z 505.055,A -85,B 0,C 180,E1 -22867.614,E2 -22867.614} C_VEL
LIN {X 0,Y 173.327,Z 495.729,A -85,B 0,C 180,E1 -22871.698,E2 -22871.698} C_VEL
LIN {X 0,Y 174.585,Z 484.818,A -85,B 0,C 180,E1 -22875.708,E2 -22875.708} C_VEL
LIN {X 0,Y 176.439,Z 472.259,A -85,B 0,C 180,E1 -22879.488,E2 -22879.488} C_VEL
LIN {X 0,Y 178.589,Z 458.77,A -85,B 0,C 180,E1 -22882.869,E2 -22882.869} C_VEL
LIN {X 0,Y 181.108,Z 444.071,A -85,B 0,C 180,E1 -22885.886,E2 -22885.886} C_VEL
LIN {X 0,Y 183.26,Z 429.68,A -85,B 0,C 180,E1 -22888.331,E2 -22888.331} C_VEL
LIN {X 0,Y 183.188,Z 426.36,A -85,B 0,C 180,E1 -22888.877,E2 -22888.877} C_VEL
LIN {X 0,Y 180.86,Z 412.265,A -85,B 0,C 180,E1 -22891.244,E2 -22891.244} C_VEL
LIN {X 0,Y 178.194,Z 398.616,A -85,B 0,C 180,E1 -22893.341,E2 -22893.341} C_VEL
LIN {X 0,Y 181.342,Z 398.96,A -85,B 0,C 180,E1 -22895.545,E2 -22895.545} C_VEL
LIN {X 0,Y 183.169,Z 400.64,A -85,B 0,C 180,E1 -22897.873,E2 -22897.873} C_VEL
LIN {X 0,Y 184.713,Z 403.117,A -85,B 0,C 180,E1 -22900.444,E2 -22900.444} C_VEL
LIN {X 0,Y 185.44,Z 406.279,A -85,B 0,C 180,E1 -22903.016,E2 -22903.016} C_VEL
LIN {X 0,Y 186.098,Z 412.053,A -85,B 0,C 180,E1 -22907.168,E2 -22907.168} C_VEL
LIN {X 0,Y 186.252,Z 414.099,A -85,B 0,C 180,E1 -22908.403,E2 -22908.403} C_VEL
LIN {X 0,Y 191.001,Z 425.584,A -85,B 0,C 180,E1 -22910.442,E2 -22910.442} C_VEL
LIN {X 0,Y 194.603,Z 437.081,A -85,B 0,C 180,E1 -22912.543,E2 -22912.543} C_VEL
LIN {X 0,Y 197.11,Z 447.723,A -85,B 0,C 180,E1 -22914.66,E2 -22914.66} C_VEL
LIN {X 0,Y 197.343,Z 449.376,A -85,B 0,C 180,E1 -22914.996,E2 -22914.996} C_VEL
LIN {X 0,Y 195.055,Z 460.799,A -85,B 0,C 180,E1 -22916.656,E2 -22916.656} C_VEL
LIN {X 0,Y 192.362,Z 471.372,A -85,B 0,C 180,E1 -22918.62,E2 -22918.62} C_VEL
LIN {X 0,Y 189.739,Z 479.943,A -85,B 0,C 180,E1 -22920.603,E2 -22920.603} C_VEL
LIN {X 0,Y 187.439,Z 487.11,A -85,B 0,C 180,E1 -22922.652,E2 -22922.652} C_VEL
LIN {X 0,Y 184.065,Z 495.973,A -85,B 0,C 180,E1 -22925.761,E2 -22925.761} C_VEL
LIN {X 0,Y 181.586,Z 502.275,A -85,B 0,C 180,E1 -22928.593,E2 -22928.593} C_VEL
LIN {X 0,Y 179.133,Z 507.839,A -85,B 0,C 180,E1 -22931.702,E2 -22931.702} C_VEL
LIN {X 0,Y 176.807,Z 512.502,A -85,B 0,C 180,E1 -22935.021,E2 -22935.021} C_VEL
LIN {X 0,Y 175.103,Z 516.041,A -85,B 0,C 180,E1 -22938.418,E2 -22938.418} C_VEL
LIN {X 0,Y 174.327,Z 517.844,A -85,B 0,C 180,E1 -22940.714,E2 -22940.714} C_VEL
LIN {X 0,Y 173.76,Z 519.211,A -85,B 0,C 180,E1 -22943.025,E2 -22943.025} C_VEL
LIN {X 0,Y 172.991,Z 520.777,A -85,B 0,C 180,E1 -22947.666,E2 -22947.666} C_VEL
LIN {X 0,Y 172.906,Z 521.001,A -85,B 0,C 180,E1 -22949.994,E2 -22949.994} C_VEL
LIN {X 0,Y 173.298,Z 520.229,A -85,B 0,C 180,E1 -22954.647,E2 -22954.647} C_VEL
LIN {X 0,Y 173.783,Z 519.279,A -85,B 0,C 180,E1 -22956.963,E2 -22956.963} C_VEL
LIN {X 0,Y 174.317,Z 517.96,A -85,B 0,C 180,E1 -22959.275,E2 -22959.275} C_VEL
LIN {X 0,Y 175.495,Z 515.173,A -85,B 0,C 180,E1 -22962.718,E2 -22962.718} C_VEL
LIN {X 0,Y 177.447,Z 511.317,A -85,B 0,C 180,E1 -22966.09,E2 -22966.09} C_VEL
LIN {X 0,Y 179.947,Z 506.3,A -85,B 0,C 180,E1 -22969.383,E2 -22969.383} C_VEL
LIN {X 0,Y 183.057,Z 498.841,A -85,B 0,C 180,E1 -22973.168,E2 -22973.168} C_VEL
LIN {X 0,Y 186.118,Z 490.739,A -85,B 0,C 180,E1 -22976.333,E2 -22976.333} C_VEL
LIN {X 0,Y 188.523,Z 484.173,A -85,B 0,C 180,E1 -22978.373,E2 -22978.373} C_VEL
LIN {X 0,Y 191.275,Z 475.389,A -85,B 0,C 180,E1 -22980.644,E2 -22980.644} C_VEL
LIN {X 0,Y 194.188,Z 464.461,A -85,B 0,C 180,E1 -22982.873,E2 -22982.873} C_VEL
LIN {X 0,Y 196.85,Z 453.148,A -85,B 0,C 180,E1 -22984.625,E2 -22984.625} C_VEL
LIN {X 0,Y 197.419,Z 450.051,A -85,B 0,C 180,E1 -22985.035,E2 -22985.035} C_VEL
LIN {X 0,Y 195.964,Z 442.205,A -85,B 0,C 180,E1 -22986.614,E2 -22986.614} C_VEL
LIN {X 0,Y 192.79,Z 430.53,A -85,B 0,C 180,E1 -22988.809,E2 -22988.809} C_VEL
LIN {X 0,Y 188.535,Z 419.19,A -85,B 0,C 180,E1 -22990.856,E2 -22990.856} C_VEL
LIN {X 0,Y 186.185,Z 413.947,A -85,B 0,C 180,E1 -22991.816,E2 -22991.816} C_VEL
LIN {X 0,Y 185.656,Z 407.925,A -85,B 0,C 180,E1 -22995.983,E2 -22995.983} C_VEL
LIN {X 0,Y 185.07,Z 402.901,A -85,B 0,C 180,E1 -22999.79,E2 -22999.79} C_VEL
LIN {X 0,Y 184.37,Z 397.77,A -85,B 0,C 180,E1 -23004.057,E2 -23004.057} C_VEL
LIN {X 0,Y 183.533,Z 392.981,A -85,B 0,C 180,E1 -23008.465,E2 -23008.465} C_VEL
LIN {X 0,Y 182.786,Z 388.982,A -85,B 0,C 180,E1 -23012.522,E2 -23012.522} C_VEL
LIN {X 0,Y 181.999,Z 385.8,A -85,B 0,C 180,E1 -23016.079,E2 -23016.079} C_VEL
LIN {X 0,Y 181.276,Z 383.186,A -85,B 0,C 180,E1 -23019.577,E2 -23019.577} C_VEL
LIN {X 0,Y 180.403,Z 379.858,A -85,B 0,C 180,E1 -23024.174,E2 -23024.174} C_VEL
LIN {X 0,Y 179.969,Z 377.553,A -85,B 0,C 180,E1 -23028.739,E2 -23028.739} C_VEL
LIN {X 0,Y 179.818,Z 376.433,A -85,B 0,C 180,E1 -23031.005,E2 -23031.005} C_VEL
LIN {X 0,Y 179.48,Z 375.445,A -85,B 0,C 180,E1 -23033.253,E2 -23033.253} C_VEL
LIN {X 0,Y 179.288,Z 373.533,A -85,B 0,C 180,E1 -23039.999,E2 -23039.999} C_VEL
LIN {X 0,Y 179.273,Z 373.404,A -85,B 0,C 180,E1 -23042.246,E2 -23042.246} C_VEL
LIN {X 0,Y 179.082,Z 373.742,A -85,B 0,C 180,E1 -23044.501,E2 -23044.501} C_VEL
LIN {X 0,Y 178.617,Z 375.766,A -85,B 0,C 180,E1 -23049.054,E2 -23049.054} C_VEL
LIN {X 0,Y 178.447,Z 380.78,A -85,B 0,C 180,E1 -23056.002,E2 -23056.002} C_VEL
LIN {X 0,Y 179.209,Z 384.362,A -85,B 0,C 180,E1 -23059.765,E2 -23059.765} C_VEL
LIN {X 0,Y 180.466,Z 391.013,A -85,B 0,C 180,E1 -23065.364,E2 -23065.364} C_VEL
LIN {X 0,Y 182.304,Z 397.237,A -85,B 0,C 180,E1 -23069.44,E2 -23069.44} C_VEL
LIN {X 0,Y 185.96,Z 409.617,A -85,B 0,C 180,E1 -23075.906,E2 -23075.906} C_VEL
LIN {X 0,Y 187.67,Z 414.511,A -85,B 0,C 180,E1 -23078.158,E2 -23078.158} C_VEL
LIN {X 0,Y 188.444,Z 419.189,A -85,B 0,C 180,E1 -23079.825,E2 -23079.825} C_VEL
LIN {X 0,Y 193.979,Z 433.857,A -85,B 0,C 180,E1 -23081.912,E2 -23081.912} C_VEL
